C09146=1141.920,201.494,-63.208,-178.121,7.460,148.864
C09147=1141.924,201.244,-63.184,-178.124,7.457,148.864
C09148=1141.929,200.995,-63.160,-178.126,7.455,148.864
C09149=1141.933,200.747,-63.136,-178.129,7.453,148.864
C09150=1141.938,200.498,-63.112,-178.132,7.450,148.865
C09151=1141.942,200.249,-63.087,-178.135,7.448,148.865
C09152=1141.947,200.000,-63.063,-178.138,7.445,148.865
C09153=1141.951,199.752,-63.038,-178.141,7.442,148.865
C09154=1141.957,199.503,-63.015,-178.143,7.441,148.866
C09155=1141.960,199.254,-62.990,-178.146,7.438,148.866
C09156=1141.965,199.005,-62.966,-178.149,7.435,148.866
C09157=1141.969,198.757,-62.942,-178.152,7.433,148.866
C09158=1141.975,198.507,-62.918,-178.154,7.430,148.866
C09159=1141.979,198.259,-62.894,-178.158,7.428,148.867
C09160=1141.983,198.010,-62.869,-178.160,7.426,148.867
C09161=1141.987,197.761,-62.845,-178.163,7.423,148.867
C09162=1141.993,197.512,-62.821,-178.165,7.421,148.867
C09163=1141.997,197.264,-62.797,-178.169,7.418,148.868
C09164=1142.001,197.015,-62.773,-178.172,7.415,148.868
C09165=1142.006,196.766,-62.750,-178.174,7.413,148.868
C09166=1142.011,196.517,-62.725,-178.177,7.411,148.868
C09167=1142.015,196.268,-62.701,-178.180,7.408,148.868
C09168=1142.020,196.019,-62.677,-178.183,7.406,148.869
C09169=1142.024,195.771,-62.653,-178.185,7.403,148.869
C09170=1142.029,195.523,-62.629,-178.188,7.402,148.869
C09171=1142.033,195.273,-62.606,-178.191,7.399,148.869
C09172=1142.038,195.025,-62.581,-178.194,7.396,148.870
C09173=1142.042,194.775,-62.558,-178.196,7.394,148.870
C09174=1142.047,194.527,-62.533,-178.200,7.391,148.870
C09175=1142.052,194.278,-62.510,-178.202,7.389,148.870
C09176=1142.056,194.029,-62.486,-178.205,7.387,148.871
C09177=1142.061,193.780,-62.463,-178.208,7.384,148.871
C09178=1142.065,193.532,-62.439,-178.210,7.382,148.871
C09179=1142.071,193.282,-62.415,-178.213,7.379,148.871
C09180=1142.075,193.034,-62.391,-178.216,7.376,148.871
C09181=1142.080,192.785,-62.367,-178.219,7.375,148.872
C09182=1142.084,192.537,-62.343,-178.222,7.372,148.872
C09183=1142.089,192.287,-62.320,-178.224,7.370,148.872
C09184=1142.093,192.039,-62.296,-178.227,7.367,148.872
C09185=1142.097,191.789,-62.272,-178.230,7.365,148.873
C09186=1142.102,191.540,-62.249,-178.233,7.362,148.873
C09187=1142.106,191.292,-62.225,-178.236,7.360,148.873
C09188=1142.111,191.043,-62.201,-178.238,7.358,148.873
C09189=1142.115,190.794,-62.177,-178.242,7.355,148.873
C09190=1142.120,190.545,-62.154,-178.244,7.353,148.874
C09191=1142.125,190.296,-62.130,-178.247,7.351,148.874
C09192=1142.129,190.048,-62.106,-178.250,7.348,148.874
C09193=1142.134,189.799,-62.083,-178.253,7.346,148.874
C09194=1142.139,189.550,-62.060,-178.256,7.343,148.875
C09195=1142.143,189.301,-62.036,-178.258,7.341,148.875
C09196=1142.148,189.052,-62.012,-178.261,7.339,148.875
C09197=1142.152,188.803,-61.989,-178.264,7.337,148.875
C09198=1142.157,188.554,-61.965,-178.267,7.334,148.876
C09199=1142.162,188.305,-61.942,-178.269,7.332,148.876
C09200=1142.166,188.057,-61.918,-178.272,7.330,148.876
C09201=1142.171,187.808,-61.895,-178.275,7.327,148.876
C09202=1142.176,187.559,-61.871,-178.278,7.325,148.877
C09203=1142.180,187.310,-61.848,-178.281,7.322,148.877
C09204=1142.184,187.061,-61.825,-178.283,7.320,148.877
C09205=1142.189,186.813,-61.802,-178.286,7.317,148.877
C09206=1142.194,186.564,-61.778,-178.289,7.316,148.878
C09207=1142.199,186.315,-61.755,-178.292,7.313,148.878
C09208=1142.203,186.066,-61.731,-178.294,7.311,148.878
C09209=1142.208,185.817,-61.708,-178.298,7.309,148.878
C09210=1142.213,185.568,-61.685,-178.300,7.306,148.879
C09211=1142.217,185.320,-61.662,-178.303,7.304,148.879
C09212=1142.221,185.071,-61.639,-178.306,7.301,148.879
C09213=1142.226,184.821,-61.615,-178.309,7.299,148.879
C09214=1142.231,184.572,-61.592,-178.311,7.296,148.880
C09215=1142.235,184.323,-61.569,-178.314,7.295,148.880
C09216=1142.240,184.075,-61.544,-178.317,7.292,148.880
C09217=1142.244,183.806,-61.520,-178.320,7.289,148.880
C09218=1142.250,183.536,-61.495,-178.323,7.287,148.881
C09219=1142.255,183.266,-61.470,-178.326,7.285,148.881
C09220=1142.260,182.996,-61.445,-178.329,7.282,148.881
C09221=1142.264,182.748,-61.422,-178.332,7.280,148.882
C09222=1142.269,182.498,-61.399,-178.335,7.278,148.882
C09223=1142.274,182.249,-61.375,-178.337,7.276,148.882
C09224=1142.278,182.000,-61.352,-178.341,7.273,148.882
C09225=1142.283,181.752,-61.330,-178.343,7.270,148.883
C09226=1142.288,181.503,-61.306,-178.346,7.268,148.883
C09227=1142.292,181.254,-61.283,-178.349,7.266,148.883
C09228=1142.296,181.006,-61.260,-178.352,7.264,148.883
C09229=1142.301,180.757,-61.237,-178.355,7.261,148.884
C09230=1142.306,180.507,-61.214,-178.357,7.259,148.884
C09231=1142.311,180.259,-61.192,-178.360,7.257,148.884
C09232=1142.315,180.010,-61.168,-178.363,7.255,148.885
C09233=1142.320,179.761,-61.145,-178.366,7.252,148.885
C09234=1142.324,179.512,-61.122,-178.369,7.250,148.885
C09235=1142.329,179.262,-61.100,-178.371,7.248,148.885
C09236=1142.334,179.014,-61.077,-178.374,7.246,148.886
C09237=1142.338,178.765,-61.054,-178.377,7.244,148.886
C09238=1142.343,178.516,-61.031,-178.380,7.241,148.886
C09239=1142.347,178.268,-61.008,-178.382,7.239,148.886
C09240=1142.352,178.018,-60.985,-178.386,7.237,148.887
C09241=1142.357,177.770,-60.963,-178.388,7.235,148.887
C09242=1142.361,177.521,-60.939,-178.391,7.232,148.887
C09243=1142.366,177.271,-60.917,-178.393,7.230,148.887
C09244=1142.370,177.023,-60.894,-178.397,7.228,148.888
C09245=1142.376,176.774,-60.871,-178.399,7.226,148.888
C09246=1142.380,176.525,-60.849,-178.402,7.223,148.888
C09247=1142.384,176.276,-60.826,-178.405,7.221,148.889
C09248=1142.389,176.028,-60.803,-178.408,7.219,148.889
C09249=1142.394,175.778,-60.781,-178.410,7.217,148.889
C09250=1142.398,175.529,-60.758,-178.414,7.214,148.889
C09251=1142.403,175.280,-60.735,-178.416,7.212,148.890
C09252=1142.408,175.032,-60.713,-178.419,7.210,148.890
C09253=1142.412,174.783,-60.689,-178.422,7.208,148.890
C09254=1142.417,174.533,-60.667,-178.425,7.206,148.891
C09255=1142.422,174.285,-60.644,-178.427,7.203,148.891
C09256=1142.426,174.036,-60.622,-178.430,7.201,148.891
C09257=1142.431,173.787,-60.599,-178.433,7.199,148.891
C09258=1142.436,173.538,-60.577,-178.436,7.197,148.892
C09259=1142.440,173.289,-60.554,-178.439,7.194,148.892
C09260=1142.445,173.040,-60.532,-178.442,7.192,148.892
C09261=1142.449,172.792,-60.509,-178.444,7.190,148.893
C09262=1142.454,172.542,-60.487,-178.447,7.188,148.893
C09263=1142.458,172.293,-60.465,-178.450,7.186,148.893
C09264=1142.464,172.044,-60.442,-178.453,7.183,148.893
C09265=1142.468,171.795,-60.420,-178.455,7.182,148.894
C09266=1142.472,171.546,-60.397,-178.459,7.179,148.894
C09267=1142.478,171.297,-60.375,-178.461,7.177,148.894
C09268=1142.482,171.048,-60.353,-178.464,7.175,148.895
C09269=1142.486,170.800,-60.330,-178.467,7.173,148.895
C09270=1142.491,170.550,-60.308,-178.469,7.171,148.895
C09271=1142.495,170.302,-60.285,-178.472,7.168,148.895
C09272=1142.500,170.053,-60.263,-178.475,7.166,148.896
C09273=1142.505,169.803,-60.240,-178.478,7.163,148.896
C09274=1142.510,169.555,-60.219,-178.481,7.162,148.896
C09275=1142.514,169.306,-60.196,-178.483,7.160,148.897
C09276=1142.519,169.056,-60.173,-178.487,7.157,148.897
C09277=1142.524,168.808,-60.152,-178.489,7.155,148.897
C09278=1142.528,168.559,-60.129,-178.492,7.153,148.898
C09279=1142.534,168.310,-60.107,-178.495,7.151,148.898
C09280=1142.538,168.061,-60.085,-178.497,7.149,148.898
C09281=1142.543,167.812,-60.063,-178.500,7.146,148.898
C09282=1142.547,167.563,-60.041,-178.503,7.145,148.899
C09283=1142.552,167.314,-60.018,-178.506,7.142,148.899
C09284=1142.557,167.065,-59.996,-178.509,7.140,148.899
C09285=1142.561,166.816,-59.974,-178.511,7.138,148.900
C09286=1142.566,166.567,-59.952,-178.515,7.136,148.900
C09287=1142.571,166.317,-59.929,-178.517,7.134,148.900
C09288=1142.576,166.069,-59.908,-178.519,7.132,148.901
C09289=1142.580,165.820,-59.885,-178.523,7.130,148.901
C09290=1142.584,165.571,-59.863,-178.525,7.128,148.901
C09291=1142.589,165.322,-59.841,-178.528,7.125,148.901
C09292=1142.594,165.073,-59.820,-178.531,7.123,148.902
C09293=1142.599,164.824,-59.797,-178.534,7.122,148.902
C09294=1142.603,164.575,-59.775,-178.537,7.119,148.903
C09295=1142.608,164.326,-59.753,-178.539,7.117,148.903
C09296=1142.613,164.077,-59.732,-178.542,7.115,148.903
C09297=1142.617,163.829,-59.710,-178.545,7.113,148.903
C09298=1142.622,163.579,-59.688,-178.548,7.111,148.904
C09299=1142.627,163.331,-59.666,-178.551,7.108,148.904
C09300=1142.631,163.081,-59.644,-178.553,7.106,148.904
C09301=1142.636,162.832,-59.622,-178.556,7.105,148.905
C09302=1142.641,162.583,-59.600,-178.559,7.102,148.905
C09303=1142.646,162.334,-59.578,-178.562,7.100,148.905
C09304=1142.650,162.085,-59.556,-178.564,7.098,148.906
C09305=1142.655,161.836,-59.534,-178.568,7.096,148.906
C09306=1142.659,161.587,-59.512,-178.570,7.094,148.906
C09307=1142.664,161.338,-59.491,-178.573,7.092,148.906
C09308=1142.669,161.090,-59.469,-178.576,7.089,148.907
C09309=1142.673,160.840,-59.447,-178.579,7.088,148.907
C09310=1142.678,160.591,-59.426,-178.581,7.086,148.908
C09311=1142.682,160.342,-59.404,-178.584,7.083,148.908
C09312=1142.687,160.093,-59.382,-178.587,7.081,148.908
C09313=1142.692,159.844,-59.360,-178.590,7.080,148.908
C09314=1142.696,159.595,-59.338,-178.593,7.077,148.909
C09315=1142.701,159.346,-59.317,-178.596,7.075,148.909
C09316=1142.706,159.096,-59.295,-178.598,7.073,148.909
C09317=1142.711,158.848,-59.274,-178.601,7.071,148.910
C09318=1142.716,158.599,-59.252,-178.604,7.069,148.910
C09319=1142.720,158.350,-59.230,-178.607,7.067,148.910
C09320=1142.725,158.101,-59.208,-178.610,7.065,148.911
C09321=1142.729,157.832,-59.186,-178.613,7.063,148.911
C09322=1142.735,157.563,-59.162,-178.615,7.060,148.911
C09323=1142.740,157.294,-59.139,-178.618,7.059,148.912
C09324=1142.745,157.025,-59.115,-178.621,7.056,148.912
C09325=1142.750,156.776,-59.094,-178.624,7.054,148.912
C09326=1142.755,156.527,-59.073,-178.627,7.052,148.913
C09327=1142.758,156.278,-59.051,-178.630,7.050,148.913
C09328=1142.764,156.029,-59.030,-178.633,7.048,148.914
C09329=1142.769,155.780,-59.009,-178.636,7.045,148.914
C09330=1142.773,155.531,-58.987,-178.638,7.044,148.914
C09331=1142.778,155.282,-58.966,-178.641,7.042,148.915
C09332=1142.783,155.033,-58.944,-178.644,7.040,148.915
C09333=1142.788,154.784,-58.922,-178.647,7.038,148.915
C09334=1142.792,154.535,-58.902,-178.649,7.036,148.915
C09335=1142.796,154.286,-58.880,-178.652,7.034,148.916
C09336=1142.802,154.037,-58.859,-178.655,7.031,148.916
C09337=1142.806,153.787,-58.837,-178.658,7.030,148.917
C09338=1142.811,153.538,-58.816,-178.661,7.028,148.917
C09339=1142.816,153.290,-58.794,-178.663,7.026,148.917
C09340=1142.820,153.041,-58.774,-178.666,7.023,148.917
C09341=1142.825,152.792,-58.752,-178.669,7.022,148.918
C09342=1142.830,152.542,-58.731,-178.672,7.020,148.918
C09343=1142.835,152.293,-58.709,-178.675,7.017,148.919
C09344=1142.839,152.044,-58.689,-178.678,7.016,148.919
C09345=1142.844,151.796,-58.667,-178.680,7.014,148.919
C09346=1142.849,151.546,-58.646,-178.683,7.012,148.920
C09347=1142.853,151.297,-58.624,-178.686,7.009,148.920
C09348=1142.858,151.048,-58.604,-178.689,7.008,148.920
C09349=1142.863,150.799,-58.583,-178.691,7.006,148.921
C09350=1142.868,150.550,-58.561,-178.694,7.004,148.921
C09351=1142.872,150.301,-58.540,-178.697,7.002,148.921
C09352=1142.877,150.052,-58.519,-178.700,7.000,148.922
C09353=1142.882,149.803,-58.498,-178.702,6.998,148.922
C09354=1142.886,149.554,-58.477,-178.705,6.996,148.922
C09355=1142.891,149.305,-58.456,-178.708,6.994,148.923
C09356=1142.896,149.056,-58.435,-178.711,6.992,148.923
C09357=1142.900,148.806,-58.414,-178.714,6.990,148.923
C09358=1142.905,148.558,-58.392,-178.716,6.989,148.924
C09359=1142.910,148.308,-58.371,-178.720,6.986,148.924
C09360=1142.915,148.059,-58.351,-178.722,6.984,148.924
C09361=1142.920,147.810,-58.330,-178.725,6.982,148.925
C09362=1142.925,147.561,-58.308,-178.727,6.981,148.925
C09363=1142.929,147.313,-58.288,-178.731,6.978,148.926
C09364=1142.934,147.063,-58.266,-178.733,6.976,148.926
C09365=1142.938,146.814,-58.246,-178.736,6.975,148.926
C09366=1142.943,146.565,-58.224,-178.739,6.973,148.927
C09367=1142.947,146.316,-58.204,-178.742,6.970,148.927
C09368=1142.953,146.067,-58.183,-178.745,6.969,148.927
C09369=1142.958,145.818,-58.162,-178.747,6.967,148.928
C09370=1142.962,145.569,-58.142,-178.750,6.965,148.928
C09371=1142.967,145.319,-58.121,-178.752,6.963,148.928
C09372=1142.971,145.071,-58.100,-178.756,6.961,148.929
C09373=1142.977,144.822,-58.079,-178.758,6.959,148.929
C09374=1142.980,144.572,-58.058,-178.761,6.957,148.930
C09375=1142.986,144.323,-58.037,-178.764,6.956,148.930
C09376=1142.990,144.074,-58.017,-178.767,6.953,148.930
C09377=1142.995,143.825,-57.996,-178.770,6.951,148.931
C09378=1143.000,143.576,-57.975,-178.772,6.949,148.931
C09379=1143.005,143.326,-57.954,-178.775,6.948,148.931
C09380=1143.009,143.077,-57.934,-178.778,6.946,148.932
C09381=1143.014,142.828,-57.913,-178.781,6.943,148.932
C09382=1143.019,142.579,-57.893,-178.784,6.942,148.932
C09383=1143.023,142.330,-57.872,-178.786,6.940,148.933
C09384=1143.028,142.081,-57.851,-178.789,6.938,148.933
C09385=1143.033,141.832,-57.831,-178.792,6.937,148.934
C09386=1143.038,141.583,-57.810,-178.795,6.934,148.934
C09387=1143.043,141.334,-57.790,-178.798,6.932,148.934
C09388=1143.047,141.085,-57.769,-178.800,6.931,148.935
C09389=1143.052,140.836,-57.748,-178.803,6.929,148.935
C09390=1143.057,140.587,-57.728,-178.805,6.927,148.935
C09391=1143.062,140.337,-57.707,-178.808,6.925,148.936
C09392=1143.066,140.089,-57.687,-178.811,6.923,148.936
C09393=1143.071,139.840,-57.666,-178.814,6.921,148.936
C09394=1143.076,139.590,-57.645,-178.817,6.919,148.937
C09395=1143.081,139.341,-57.626,-178.820,6.917,148.937
C09396=1143.085,139.092,-57.605,-178.822,6.916,148.938
C09397=1143.090,138.843,-57.584,-178.825,6.914,148.938
C09398=1143.095,138.594,-57.564,-178.828,6.912,148.938
C09399=1143.099,138.345,-57.543,-178.831,6.910,148.939
C09400=1143.104,138.095,-57.522,-178.834,6.908,148.939
C09401=1143.109,137.846,-57.503,-178.837,6.906,148.940
C09402=1143.113,137.597,-57.482,-178.839,6.905,148.940
C09403=1143.118,137.348,-57.462,-178.842,6.903,148.940
C09404=1143.123,137.099,-57.441,-178.845,6.901,148.941
C09405=1143.128,136.850,-57.421,-178.848,6.899,148.941
C09406=1143.133,136.601,-57.401,-178.851,6.897,148.941
C09407=1143.138,136.352,-57.380,-178.853,6.895,148.942
C09408=1143.142,136.103,-57.360,-178.856,6.893,148.942
C09409=1143.147,135.853,-57.340,-178.858,6.892,148.942
C09410=1143.152,135.604,-57.320,-178.861,6.890,148.943
C09411=1143.156,135.355,-57.300,-178.864,6.887,148.943
C09412=1143.161,135.106,-57.279,-178.867,6.886,148.944
C09413=1143.166,134.856,-57.259,-178.870,6.884,148.944
C09414=1143.170,134.607,-57.239,-178.873,6.882,148.944
C09415=1143.176,134.359,-57.219,-178.875,6.881,148.945
C09416=1143.180,134.110,-57.199,-178.878,6.879,148.945
C09417=1143.185,133.860,-57.178,-178.881,6.877,148.946
C09418=1143.190,133.611,-57.158,-178.884,6.875,148.946
C09419=1143.195,133.362,-57.138,-178.887,6.873,148.946
C09420=1143.199,133.112,-57.118,-178.889,6.871,148.947
C09421=1143.204,132.864,-57.098,-178.892,6.870,148.947
C09422=1143.209,132.615,-57.078,-178.895,6.868,148.948
C09423=1143.214,132.365,-57.058,-178.898,6.866,148.948
C09424=1143.219,132.116,-57.037,-178.900,6.864,148.948
C09425=1143.224,131.848,-57.016,-178.904,6.862,148.949
C09426=1143.229,131.579,-56.995,-178.906,6.860,148.949
C09427=1143.234,131.311,-56.973,-178.909,6.859,148.949
C09428=1143.239,131.042,-56.952,-178.912,6.856,148.950
C09429=1143.243,130.792,-56.932,-178.915,6.854,148.950
C09430=1143.249,130.544,-56.912,-178.918,6.853,148.951
C09431=1143.254,130.294,-56.892,-178.921,6.851,148.951
C09432=1143.258,130.045,-56.871,-178.923,6.849,148.951
C09433=1143.263,129.796,-56.852,-178.926,6.848,148.952
C09434=1143.268,129.547,-56.831,-178.929,6.846,148.952
C09435=1143.273,129.298,-56.812,-178.931,6.844,148.953
C09436=1143.278,129.048,-56.793,-178.935,6.842,148.953
C09437=1143.282,128.799,-56.772,-178.937,6.840,148.953
C09438=1143.287,128.550,-56.752,-178.940,6.838,148.954
C09439=1143.292,128.302,-56.732,-178.943,6.837,148.954
C09440=1143.297,128.052,-56.713,-178.946,6.835,148.955
C09441=1143.301,127.802,-56.693,-178.949,6.834,148.955
C09442=1143.306,127.553,-56.673,-178.952,6.832,148.956
C09443=1143.311,127.305,-56.653,-178.954,6.830,148.956
C09444=1143.316,127.055,-56.634,-178.957,6.828,148.956
C09445=1143.320,126.806,-56.613,-178.960,6.827,148.957
C09446=1143.326,126.557,-56.594,-178.962,6.825,148.957
C09447=1143.330,126.308,-56.575,-178.965,6.823,148.958
C09448=1143.335,126.058,-56.555,-178.968,6.822,148.958
C09449=1143.339,125.809,-56.535,-178.971,6.819,148.958
C09450=1143.344,125.561,-56.516,-178.974,6.817,148.959
C09451=1143.349,125.311,-56.496,-178.977,6.816,148.959
C09452=1143.354,125.061,-56.476,-178.979,6.814,148.960
C09453=1143.359,124.813,-56.456,-178.982,6.812,148.960
C09454=1143.364,124.564,-56.437,-178.985,6.811,148.960
C09455=1143.368,124.314,-56.417,-178.987,6.809,148.961
C09456=1143.374,124.065,-56.398,-178.990,6.807,148.961
C09457=1143.378,123.816,-56.378,-178.993,6.806,148.962
C09458=1143.382,123.566,-56.359,-178.996,6.804,148.962
C09459=1143.387,123.318,-56.339,-178.998,6.802,148.962
C09460=1143.392,123.069,-56.319,-179.001,6.800,148.963
C09461=1143.397,122.819,-56.300,-179.004,6.799,148.963
C09462=1143.402,122.570,-56.281,-179.007,6.797,148.964
C09463=1143.407,122.321,-56.261,-179.009,6.795,148.964
C09464=1143.412,122.072,-56.242,-179.012,6.794,148.964
C09465=1143.416,121.822,-56.223,-179.015,6.792,148.965
C09466=1143.421,121.573,-56.203,-179.017,6.790,148.965
C09467=1143.426,121.324,-56.184,-179.020,6.789,148.966
C09468=1143.431,121.074,-56.164,-179.023,6.787,148.966
C09469=1143.435,120.825,-56.145,-179.026,6.785,148.966
C09470=1143.440,120.576,-56.126,-179.029,6.783,148.967
C09471=1143.445,120.327,-56.106,-179.032,6.781,148.967
C09472=1143.451,120.078,-56.087,-179.035,6.780,148.968
C09473=1143.455,119.829,-56.068,-179.038,6.778,148.968
C09474=1143.460,119.580,-56.048,-179.040,6.776,148.969
C09475=1143.465,119.330,-56.029,-179.043,6.775,148.969
C09476=1143.469,119.081,-56.009,-179.046,6.773,148.969
C09477=1143.474,118.832,-55.990,-179.048,6.771,148.970
C09478=1143.479,118.582,-55.971,-179.051,6.770,148.970
C09479=1143.484,118.334,-55.951,-179.054,6.768,148.971
C09480=1143.488,118.084,-55.932,-179.057,6.766,148.971
C09481=1143.493,117.835,-55.913,-179.059,6.764,148.971
C09482=1143.498,117.586,-55.893,-179.062,6.763,148.972
C09483=1143.503,117.337,-55.875,-179.065,6.761,148.972
C09484=1143.508,117.087,-55.856,-179.068,6.759,148.973
C09485=1143.513,116.838,-55.836,-179.071,6.758,148.973
C09486=1143.517,116.589,-55.817,-179.073,6.756,148.974
C09487=1143.523,116.340,-55.798,-179.076,6.755,148.974
C09488=1143.527,116.091,-55.778,-179.079,6.753,148.974
C09489=1143.532,115.842,-55.760,-179.082,6.751,148.975
C09490=1143.537,115.592,-55.741,-179.084,6.750,148.975
C09491=1143.542,115.343,-55.721,-179.087,6.748,148.976
C09492=1143.546,115.094,-55.702,-179.090,6.746,148.976
C09493=1143.552,114.845,-55.683,-179.093,6.745,148.977
C09494=1143.556,114.595,-55.665,-179.095,6.743,148.977
C09495=1143.561,114.346,-55.645,-179.098,6.741,148.977
C09496=1143.565,114.097,-55.626,-179.101,6.739,148.978
C09497=1143.571,113.848,-55.607,-179.104,6.738,148.978
C09498=1143.576,113.598,-55.588,-179.107,6.736,148.979
C09499=1143.580,113.349,-55.569,-179.109,6.736,148.979
C09500=1143.585,113.100,-55.550,-179.112,6.734,148.980
C09501=1143.590,112.850,-55.532,-179.114,6.732,148.980
C09502=1143.595,112.601,-55.512,-179.117,6.730,148.980
C09503=1143.599,112.352,-55.493,-179.120,6.729,148.981
C09504=1143.605,112.103,-55.475,-179.122,6.727,148.981
C09505=1143.609,111.854,-55.456,-179.125,6.725,148.982
C09506=1143.614,111.605,-55.437,-179.128,6.724,148.982
C09507=1143.619,111.355,-55.418,-179.131,6.722,148.983
C09508=1143.624,111.106,-55.399,-179.134,6.721,148.983
C09509=1143.629,110.857,-55.381,-179.137,6.719,148.983
C09510=1143.634,110.607,-55.361,-179.139,6.717,148.984
C09511=1143.639,110.358,-55.343,-179.142,6.716,148.984
C09512=1143.643,110.109,-55.324,-179.145,6.714,148.985
C09513=1143.648,109.860,-55.305,-179.147,6.712,148.985
C09514=1143.654,109.610,-55.286,-179.150,6.711,148.986
C09515=1143.658,109.361,-55.267,-179.153,6.709,148.986
C09516=1143.662,109.112,-55.249,-179.156,6.708,148.987
C09517=1143.668,108.863,-55.230,-179.159,6.706,148.987
C09518=1143.672,108.613,-55.212,-179.162,6.704,148.987
C09519=1143.677,108.364,-55.192,-179.164,6.703,148.988
C09520=1143.682,108.115,-55.174,-179.166,6.702,148.988
C09521=1143.686,107.866,-55.155,-179.169,6.700,148.989
C09522=1143.692,107.617,-55.137,-179.172,6.698,148.989
C09523=1143.696,107.367,-55.118,-179.175,6.697,148.990
C09524=1143.701,107.118,-55.100,-179.178,6.695,148.990
C09525=1143.707,106.869,-55.081,-179.181,6.694,148.990
C09526=1143.711,106.619,-55.062,-179.183,6.692,148.991
C09527=1143.716,106.370,-55.044,-179.186,6.690,148.991
C09528=1143.721,106.121,-55.026,-179.189,6.689,148.992
C09529=1143.726,105.853,-55.005,-179.192,6.687,148.992
C09530=1143.731,105.584,-54.985,-179.195,6.686,148.993
C09531=1143.736,105.316,-54.966,-179.197,6.684,148.993
C09532=1143.742,105.047,-54.946,-179.200,6.682,148.994
C09533=1143.747,104.798,-54.927,-179.203,6.681,148.994
C09534=1143.751,104.549,-54.909,-179.206,6.679,148.995
C09535=1143.757,104.299,-54.890,-179.209,6.677,148.995
C09536=1143.761,104.050,-54.871,-179.212,6.676,148.995
C09537=1143.766,103.801,-54.853,-179.214,6.674,148.996
C09538=1143.770,103.551,-54.835,-179.217,6.672,148.996
C09539=1143.776,103.303,-54.816,-179.220,6.671,148.997
C09540=1143.781,103.053,-54.798,-179.223,6.669,148.997
C09541=1143.786,102.804,-54.780,-179.225,6.669,148.998
C09542=1143.790,102.554,-54.761,-179.228,6.667,148.998
C09543=1143.796,102.305,-54.743,-179.231,6.665,148.999
C09544=1143.800,102.056,-54.724,-179.233,6.663,148.999
C09545=1143.805,101.807,-54.706,-179.236,6.662,148.999
C09546=1143.809,101.557,-54.688,-179.239,6.660,149.000
C09547=1143.814,101.308,-54.670,-179.242,6.659,149.000
C09548=1143.820,101.059,-54.651,-179.245,6.657,149.001
C09549=1143.825,100.809,-54.633,-179.247,6.655,149.001
C09550=1143.829,100.561,-54.615,-179.250,6.655,149.002
C09551=1143.834,100.311,-54.596,-179.252,6.653,149.002
C09552=1143.839,100.062,-54.578,-179.256,6.652,149.003
C09553=1143.844,99.813,-54.560,-179.258,6.650,149.003
C09554=1143.849,99.563,-54.542,-179.261,6.648,149.004
C09555=1143.854,99.314,-54.524,-179.264,6.647,149.004
C09556=1143.858,99.064,-54.505,-179.267,6.645,149.004
C09557=1143.863,98.815,-54.487,-179.269,6.644,149.005
C09558=1143.868,98.566,-54.469,-179.272,6.643,149.005
C09559=1143.873,98.317,-54.451,-179.275,6.641,149.006
C09560=1143.878,98.067,-54.433,-179.277,6.639,149.006
C09561=1143.883,97.818,-54.416,-179.280,6.638,149.007
C09562=1143.887,97.568,-54.397,-179.283,6.636,149.007
C09563=1143.892,97.319,-54.379,-179.286,6.635,149.008
C09564=1143.897,97.070,-54.361,-179.288,6.634,149.008
C09565=1143.903,96.820,-54.343,-179.291,6.632,149.009
C09566=1143.908,96.571,-54.325,-179.294,6.630,149.009
C09567=1143.913,96.322,-54.307,-179.296,6.629,149.009
C09568=1143.918,96.073,-54.289,-179.300,6.627,149.010
C09569=1143.922,95.824,-54.271,-179.302,6.626,149.011
C09570=1143.927,95.574,-54.252,-179.305,6.624,149.011
C09571=1143.932,95.325,-54.234,-179.307,6.623,149.011
C09572=1143.937,95.076,-54.216,-179.310,6.622,149.012
C09573=1143.942,94.826,-54.198,-179.313,6.620,149.012
C09574=1143.946,94.577,-54.180,-179.316,6.619,149.013
C09575=1143.951,94.328,-54.162,-179.319,6.617,149.013
C09576=1143.956,94.079,-54.144,-179.321,6.616,149.014
C09577=1143.961,93.829,-54.127,-179.323,6.614,149.014
C09578=1143.966,93.580,-54.109,-179.326,6.613,149.015
C09579=1143.971,93.331,-54.091,-179.329,6.611,149.015
C09580=1143.976,93.082,-54.073,-179.332,6.610,149.016
C09581=1143.980,92.833,-54.056,-179.335,6.608,149.016
C09582=1143.986,92.583,-54.039,-179.337,6.607,149.016
C09583=1143.990,92.333,-54.020,-179.340,6.606,149.017
C09584=1143.995,92.084,-54.002,-179.343,6.604,149.017
C09585=1144.000,91.835,-53.984,-179.346,6.602,149.018
C09586=1144.005,91.585,-53.966,-179.348,6.601,149.018
C09587=1144.010,91.336,-53.949,-179.351,6.600,149.019
C09588=1144.015,91.086,-53.931,-179.354,6.599,149.019
C09589=1144.020,90.837,-53.913,-179.357,6.597,149.020
C09590=1144.025,90.588,-53.895,-179.359,6.595,149.020
C09591=1144.029,90.339,-53.878,-179.362,6.594,149.021
C09592=1144.034,90.089,-53.860,-179.364,6.593,149.021
C09593=1144.039,89.840,-53.843,-179.367,6.591,149.022
C09594=1144.044,89.591,-53.825,-179.370,6.590,149.022
C09595=1144.049,89.341,-53.807,-179.373,6.588,149.023
C09596=1144.054,89.092,-53.789,-179.376,6.586,149.023
C09597=1144.059,88.842,-53.772,-179.378,6.586,149.024
C09598=1144.063,88.594,-53.755,-179.381,6.584,149.024
C09599=1144.068,88.344,-53.737,-179.384,6.583,149.024
C09600=1144.073,88.095,-53.719,-179.386,6.581,149.025
C09601=1144.078,87.845,-53.701,-179.389,6.579,149.025
C09602=1144.084,87.596,-53.684,-179.392,6.579,149.026
C09603=1144.088,87.347,-53.667,-179.395,6.577,149.026
C09604=1144.094,87.098,-53.650,-179.397,6.575,149.027
C09605=1144.099,86.848,-53.632,-179.400,6.574,149.027
C09606=1144.103,86.599,-53.614,-179.403,6.573,149.028
C09607=1144.108,86.350,-53.597,-179.405,6.572,149.028
C09608=1144.113,86.101,-53.579,-179.408,6.570,149.029
C09609=1144.118,85.851,-53.562,-179.411,6.568,149.029
C09610=1144.123,85.602,-53.544,-179.413,6.568,149.030
C09611=1144.127,85.352,-53.527,-179.416,6.566,149.030
C09612=1144.132,85.103,-53.509,-179.419,6.564,149.031
C09613=1144.138,84.853,-53.492,-179.422,6.563,149.031
C09614=1144.142,84.604,-53.475,-179.425,6.561,149.032
C09615=1144.147,84.355,-53.457,-179.427,6.561,149.032
C09616=1144.152,84.105,-53.440,-179.430,6.559,149.033
C09617=1144.158,83.856,-53.423,-179.433,6.557,149.033
C09618=1144.162,83.607,-53.406,-179.435,6.555,149.033
C09619=1144.167,83.358,-53.388,-179.438,6.555,149.034
C09620=1144.172,83.108,-53.371,-179.441,6.553,149.035
C09621=1144.176,82.859,-53.353,-179.443,6.552,149.035
C09622=1144.182,82.609,-53.336,-179.446,6.551,149.035
C09623=1144.186,82.360,-53.319,-179.449,6.549,149.036
C09624=1144.191,82.110,-53.301,-179.452,6.548,149.036
C09625=1144.197,81.861,-53.284,-179.454,6.546,149.037
C09626=1144.201,81.612,-53.268,-179.457,6.546,149.038
C09627=1144.206,81.363,-53.250,-179.460,6.544,149.038
C09628=1144.211,81.113,-53.233,-179.462,6.542,149.038
C09629=1144.216,80.863,-53.216,-179.465,6.541,149.039
C09630=1144.221,80.614,-53.198,-179.468,6.540,149.039
C09631=1144.226,80.365,-53.182,-179.470,6.539,149.040
C09632=1144.231,80.116,-53.164,-179.473,6.537,149.040
C09633=1144.237,79.847,-53.146,-179.476,6.535,149.041
C09634=1144.242,79.579,-53.128,-179.479,6.534,149.041
C09635=1144.247,79.311,-53.108,-179.482,6.532,149.042
C09636=1144.252,79.042,-53.090,-179.485,6.531,149.042
C09637=1144.257,78.793,-53.073,-179.487,6.530,149.043
C09638=1144.263,78.543,-53.056,-179.490,6.528,149.043
C09639=1144.267,78.294,-53.040,-179.493,6.527,149.044
C09640=1144.272,78.045,-53.022,-179.495,6.526,149.044
C09641=1144.276,77.795,-53.005,-179.498,6.525,149.045
C09642=1144.282,77.546,-52.988,-179.501,6.523,149.045
C09643=1144.287,77.297,-52.971,-179.504,6.522,149.046
C09644=1144.292,77.047,-52.954,-179.506,6.521,149.046
C09645=1144.296,76.797,-52.937,-179.509,6.519,149.047
C09646=1144.302,76.548,-52.921,-179.512,6.518,149.047
C09647=1144.306,76.299,-52.903,-179.514,6.517,149.048
C09648=1144.311,76.050,-52.886,-179.517,6.515,149.048
C09649=1144.316,75.800,-52.869,-179.520,6.514,149.049
C09650=1144.321,75.551,-52.853,-179.523,6.513,149.049
C09651=1144.326,75.301,-52.836,-179.525,6.511,149.050
C09652=1144.331,75.052,-52.819,-179.528,6.510,149.050
C09653=1144.336,74.802,-52.802,-179.530,6.509,149.051
C09654=1144.341,74.553,-52.785,-179.533,6.508,149.051
C09655=1144.346,74.304,-52.769,-179.536,6.506,149.052
C09656=1144.351,74.054,-52.751,-179.538,6.505,149.052
C09657=1144.356,73.805,-52.735,-179.541,6.504,149.053
C09658=1144.361,73.556,-52.718,-179.544,6.502,149.053
C09659=1144.366,73.306,-52.701,-179.546,6.501,149.054
C09660=1144.371,73.057,-52.685,-179.549,6.500,149.054
C09661=1144.376,72.807,-52.668,-179.552,6.498,149.055
C09662=1144.380,72.558,-52.651,-179.555,6.497,149.055
C09663=1144.386,72.309,-52.634,-179.557,6.496,149.056
C09664=1144.391,72.059,-52.617,-179.560,6.495,149.056
C09665=1144.395,71.810,-52.601,-179.563,6.494,149.057
C09666=1144.401,71.561,-52.584,-179.565,6.492,149.057
C09667=1144.406,71.311,-52.567,-179.569,6.491,149.058
C09668=1144.410,71.062,-52.551,-179.571,6.490,149.058
C09669=1144.416,70.813,-52.534,-179.573,6.488,149.059
C09670=1144.420,70.563,-52.517,-179.576,6.487,149.059
C09671=1144.425,70.314,-52.500,-179.579,6.486,149.060
C09672=1144.430,70.064,-52.485,-179.582,6.484,149.060
C09673=1144.435,69.815,-52.467,-179.584,6.483,149.061
C09674=1144.440,69.565,-52.451,-179.587,6.482,149.061
C09675=1144.445,69.316,-52.434,-179.590,6.481,149.062
C09676=1144.450,69.067,-52.417,-179.592,6.479,149.062
C09677=1144.455,68.818,-52.401,-179.595,6.478,149.063
C09678=1144.460,68.568,-52.385,-179.598,6.477,149.063
C09679=1144.465,68.318,-52.368,-179.601,6.475,149.064
C09680=1144.470,68.069,-52.351,-179.603,6.474,149.064
C09681=1144.475,67.820,-52.335,-179.606,6.473,149.065
C09682=1144.480,67.571,-52.318,-179.608,6.472,149.065
C09683=1144.485,67.321,-52.302,-179.611,6.470,149.066
C09684=1144.489,67.071,-52.286,-179.614,6.469,149.066
C09685=1144.495,66.822,-52.269,-179.616,6.468,149.067
C09686=1144.499,66.573,-52.252,-179.619,6.467,149.067
C09687=1144.505,66.323,-52.237,-179.622,6.465,149.068
C09688=1144.509,66.074,-52.220,-179.624,6.465,149.068
C09689=1144.514,65.825,-52.204,-179.627,6.463,149.069
C09690=1144.519,65.575,-52.188,-179.630,6.462,149.069
C09691=1144.524,65.325,-52.170,-179.633,6.461,149.070
C09692=1144.530,65.076,-52.154,-179.635,6.459,149.070
C09693=1144.534,64.826,-52.138,-179.638,6.459,149.071
C09694=1144.539,64.577,-52.122,-179.641,6.457,149.071
C09695=1144.544,64.328,-52.105,-179.643,6.456,149.072
C09696=1144.549,64.078,-52.090,-179.646,6.454,149.072
C09697=1144.554,63.829,-52.073,-179.649,6.453,149.073
C09698=1144.560,63.580,-52.056,-179.651,6.452,149.073
C09699=1144.564,63.330,-52.040,-179.654,6.451,149.074
C09700=1144.569,63.081,-52.024,-179.656,6.450,149.074
C09701=1144.574,62.831,-52.008,-179.659,6.449,149.075
C09702=1144.579,62.582,-51.992,-179.662,6.447,149.075
C09703=1144.584,62.332,-51.976,-179.664,6.446,149.076
C09704=1144.589,62.083,-51.959,-179.667,6.445,149.076
C09705=1144.594,61.834,-51.943,-179.669,6.444,149.077
C09706=1144.599,61.584,-51.927,-179.673,6.443,149.078
C09707=1144.604,61.335,-51.910,-179.675,6.441,149.078
C09708=1144.609,61.085,-51.895,-179.678,6.440,149.078
C09709=1144.613,60.836,-51.878,-179.681,6.439,149.079
C09710=1144.619,60.587,-51.862,-179.683,6.438,149.079
C09711=1144.623,60.337,-51.846,-179.686,6.436,149.080
C09712=1144.629,60.088,-51.830,-179.689,6.435,149.081
C09713=1144.634,59.839,-51.814,-179.691,6.434,149.081
C09714=1144.638,59.589,-51.798,-179.694,6.433,149.081
C09715=1144.644,59.339,-51.782,-179.696,6.432,149.082
C09716=1144.648,59.090,-51.766,-179.699,6.430,149.083
C09717=1144.654,58.841,-51.750,-179.701,6.430,149.083
C09718=1144.658,58.591,-51.733,-179.705,6.428,149.084
C09719=1144.664,58.342,-51.718,-179.707,6.427,149.084
C09720=1144.669,58.093,-51.702,-179.709,6.426,149.085
C09721=1144.673,57.843,-51.686,-179.713,6.425,149.085
C09722=1144.679,57.593,-51.670,-179.715,6.424,149.086
C09723=1144.683,57.344,-51.653,-179.718,6.422,149.086
C09724=1144.689,57.094,-51.638,-179.720,6.422,149.087
C09725=1144.694,56.845,-51.622,-179.723,6.420,149.087
C09726=1144.699,56.596,-51.606,-179.725,6.419,149.088
C09727=1144.704,56.346,-51.590,-179.728,6.418,149.088
C09728=1144.709,56.096,-51.574,-179.731,6.416,149.089
C09729=1144.714,55.847,-51.558,-179.733,6.415,149.089
C09730=1144.719,55.598,-51.542,-179.737,6.414,149.090
C09731=1144.723,55.348,-51.527,-179.739,6.413,149.090
C09732=1144.729,55.099,-51.511,-179.742,6.412,149.091
C09733=1144.734,54.850,-51.495,-179.744,6.411,149.091
C09734=1144.739,54.600,-51.479,-179.747,6.409,149.092
C09735=1144.744,54.350,-51.463,-179.749,6.409,149.092
C09736=1144.749,54.101,-51.448,-179.752,6.407,149.093
C09737=1144.754,53.832,-51.430,-179.755,6.406,149.093
C09738=1144.760,53.563,-51.413,-179.758,6.405,149.094
C09739=1144.765,53.295,-51.396,-179.761,6.404,149.095
C09740=1144.770,53.027,-51.380,-179.764,6.402,149.095
C09741=1144.776,52.777,-51.364,-179.766,6.401,149.096
C09742=1144.780,52.528,-51.348,-179.769,6.400,149.096
C09743=1144.785,52.278,-51.332,-179.771,6.399,149.097
C09744=1144.791,52.029,-51.316,-179.774,6.398,149.097
C09745=1144.795,51.779,-51.301,-179.777,6.397,149.098
C09746=1144.800,51.530,-51.285,-179.779,6.395,149.098
C09747=1144.806,51.280,-51.270,-179.782,6.395,149.099
C09748=1144.810,51.030,-51.254,-179.785,6.393,149.099
C09749=1144.816,50.782,-51.238,-179.787,6.393,149.100
C09750=1144.820,50.532,-51.223,-179.790,6.391,149.100
C09751=1144.826,50.283,-51.207,-179.792,6.390,149.101
C09752=1144.830,50.033,-51.191,-179.795,6.389,149.101
C09753=1144.836,49.784,-51.176,-179.798,6.388,149.102
C09754=1144.840,49.534,-51.161,-179.800,6.387,149.102
C09755=1144.846,49.285,-51.145,-179.803,6.386,149.103
C09756=1144.851,49.035,-51.129,-179.806,6.385,149.104
C09757=1144.855,48.786,-51.114,-179.808,6.384,149.104
C09758=1144.861,48.536,-51.098,-179.811,6.382,149.105
C09759=1144.865,48.286,-51.082,-179.813,6.382,149.105
C09760=1144.870,48.037,-51.067,-179.816,6.380,149.106
C09761=1144.875,47.788,-51.052,-179.819,6.379,149.106
C09762=1144.881,47.538,-51.036,-179.821,6.378,149.107
C09763=1144.885,47.289,-51.021,-179.824,6.377,149.107
C09764=1144.890,47.039,-51.005,-179.827,6.376,149.108
C09765=1144.896,46.790,-50.990,-179.829,6.375,149.108
C09766=1144.900,46.541,-50.975,-179.832,6.374,149.109
C09767=1144.906,46.291,-50.959,-179.834,6.373,149.109
C09768=1144.911,46.042,-50.944,-179.837,6.371,149.110
C09769=1144.915,45.792,-50.928,-179.840,6.371,149.111
C09770=1144.920,45.543,-50.913,-179.843,6.369,149.111
C09771=1144.926,45.293,-50.897,-179.845,6.368,149.111
C09772=1144.931,45.044,-50.883,-179.848,6.367,149.112
C09773=1144.936,44.794,-50.867,-179.850,6.366,149.113
C09774=1144.940,44.544,-50.852,-179.853,6.364,149.113
C09775=1144.946,44.295,-50.836,-179.856,6.364,149.114
C09776=1144.951,44.046,-50.821,-179.858,6.362,149.114
C09777=1144.956,43.797,-50.806,-179.861,6.362,149.115
C09778=1144.961,43.547,-50.790,-179.864,6.360,149.115
C09779=1144.966,43.297,-50.776,-179.866,6.359,149.116
C09780=1144.971,43.047,-50.760,-179.868,6.359,149.116
C09781=1144.975,42.798,-50.745,-179.871,6.357,149.117
C09782=1144.981,42.549,-50.729,-179.874,6.357,149.117
C09783=1144.986,42.300,-50.714,-179.877,6.355,149.118
C09784=1144.991,42.050,-50.699,-179.879,6.354,149.118
C09785=1144.997,41.800,-50.684,-179.882,6.353,149.119
C09786=1145.001,41.551,-50.669,-179.884,6.352,149.119
C09787=1145.007,41.302,-50.653,-179.887,6.351,149.120
C09788=1145.011,41.051,-50.639,-179.890,6.350,149.121
C09789=1145.016,40.802,-50.623,-179.892,6.349,149.121
C09790=1145.021,40.553,-50.608,-179.895,6.348,149.122
C09791=1145.026,40.304,-50.592,-179.897,6.347,149.122
C09792=1145.031,40.054,-50.578,-179.900,6.346,149.123
C09793=1145.037,39.804,-50.563,-179.903,6.345,149.123
C09794=1145.041,39.555,-50.548,-179.905,6.343,149.124
C09795=1145.046,39.306,-50.533,-179.908,6.343,149.124
C09796=1145.052,39.056,-50.518,-179.911,6.341,149.125
C09797=1145.056,38.807,-50.503,-179.913,6.341,149.125
C09798=1145.062,38.557,-50.488,-179.916,6.340,149.126
C09799=1145.067,38.308,-50.473,-179.918,6.338,149.126
C09800=1145.072,38.058,-50.457,-179.920,6.338,149.127
C09801=1145.076,37.808,-50.443,-179.924,6.336,149.128
C09802=1145.082,37.559,-50.427,-179.926,6.335,149.128
C09803=1145.087,37.309,-50.413,-179.929,6.335,149.129
C09804=1145.091,37.060,-50.398,-179.931,6.333,149.129
C09805=1145.097,36.810,-50.383,-179.933,6.333,149.130
C09806=1145.102,36.561,-50.368,-179.937,6.331,149.130
C09807=1145.107,36.311,-50.352,-179.939,6.330,149.131
C09808=1145.112,36.062,-50.338,-179.942,6.329,149.131
C09809=1145.117,35.813,-50.323,-179.944,6.328,149.132
C09810=1145.122,35.563,-50.308,-179.946,6.328,149.132
C09811=1145.127,35.314,-50.293,-179.950,6.326,149.133
C09812=1145.132,35.064,-50.279,-179.952,6.325,149.133
C09813=1145.137,34.814,-50.263,-179.955,6.324,149.134
C09814=1145.142,34.565,-50.249,-179.957,6.323,149.134
C09815=1145.147,34.316,-50.234,-179.959,6.323,149.135
C09816=1145.153,34.066,-50.219,-179.963,6.321,149.136
C09817=1145.157,33.817,-50.204,-179.965,6.320,149.136
C09818=1145.162,33.567,-50.190,-179.968,6.319,149.137
C09819=1145.168,33.317,-50.174,-179.970,6.318,149.137
C09820=1145.173,33.068,-50.160,-179.972,6.317,149.138
C09821=1145.178,32.818,-50.146,-179.976,6.316,149.138
C09822=1145.183,32.569,-50.130,-179.978,6.315,149.139
C09823=1145.188,32.319,-50.116,-179.980,6.315,149.139
C09824=1145.193,32.070,-50.101,-179.983,6.313,149.140
C09825=1145.198,31.820,-50.087,-179.985,6.312,149.140
C09826=1145.204,31.571,-50.072,-179.989,6.311,149.141
C09827=1145.209,31.322,-50.057,-179.991,6.310,149.141
C09828=1145.214,31.072,-50.043,-179.993,6.310,149.142
C09829=1145.218,30.823,-50.028,-179.996,6.308,149.143
C09830=1145.224,30.573,-50.013,-179.998,6.307,149.143
C09831=1145.229,30.323,-49.999,179.998,6.306,149.144
C09832=1145.233,30.074,-49.984,179.996,6.305,149.144
C09833=1145.238,29.824,-49.969,179.994,6.305,149.145
C09834=1145.243,29.575,-49.955,179.991,6.303,149.145
C09835=1145.249,29.325,-49.940,179.989,6.302,149.146
C09836=1145.254,29.075,-49.925,179.986,6.302,149.146
C09837=1145.259,28.826,-49.911,179.983,6.300,149.147
C09838=1145.264,28.576,-49.897,179.981,6.300,149.148
C09839=1145.269,28.328,-49.882,179.978,6.299,149.148
C09840=1145.275,28.078,-49.867,179.976,6.297,149.148
C09841=1145.280,27.809,-49.852,179.973,6.297,149.149
C09842=1145.285,27.539,-49.837,179.970,6.296,149.150
C09843=1145.290,27.271,-49.821,179.968,6.295,149.150
C09844=1145.296,27.002,-49.805,179.964,6.294,149.151
C09845=1145.301,26.752,-49.790,179.962,6.293,149.151
C09846=1145.306,26.502,-49.776,179.959,6.292,149.152
C09847=1145.312,26.253,-49.762,179.957,6.291,149.153
C09848=1145.317,26.003,-49.748,179.955,6.290,149.153
C09849=1145.321,25.754,-49.733,179.951,6.289,149.154
C09850=1145.326,25.505,-49.718,179.949,6.288,149.154
C09851=1145.331,25.255,-49.704,179.947,6.287,149.155
C09852=1145.336,25.005,-49.690,179.944,6.286,149.155
C09853=1145.342,24.756,-49.675,179.941,6.285,149.156
C09854=1145.347,24.506,-49.661,179.939,6.285,149.156
C09855=1145.352,24.256,-49.647,179.936,6.283,149.157
C09856=1145.357,24.007,-49.632,179.934,6.282,149.158
C09857=1145.362,23.758,-49.618,179.931,6.282,149.158
C09858=1145.367,23.508,-49.603,179.928,6.280,149.159
C09859=1145.372,23.259,-49.589,179.926,6.280,149.159
C09860=1145.377,23.009,-49.575,179.924,6.279,149.160
C09861=1145.382,22.760,-49.561,179.921,6.277,149.160
C09862=1145.387,22.510,-49.547,179.918,6.277,149.161
C09863=1145.392,22.260,-49.532,179.916,6.276,149.161
C09864=1145.398,22.011,-49.518,179.913,6.275,149.162
C09865=1145.403,21.761,-49.504,179.911,6.274,149.162
C09866=1145.408,21.512,-49.490,179.908,6.273,149.163
C09867=1145.413,21.262,-49.476,179.906,6.272,149.163
C09868=1145.418,21.013,-49.462,179.903,6.271,149.164
C09869=1145.423,20.763,-49.447,179.901,6.270,149.165
C09870=1145.428,20.514,-49.433,179.898,6.270,149.165
C09871=1145.433,20.264,-49.419,179.895,6.268,149.166
C09872=1145.439,20.015,-49.405,179.893,6.268,149.166
C09873=1145.444,19.765,-49.391,179.890,6.267,149.167
C09874=1145.448,19.515,-49.376,179.888,6.265,149.167
C09875=1145.453,19.266,-49.362,179.885,6.265,149.168
C09876=1145.459,19.017,-49.348,179.883,6.264,149.168
C09877=1145.464,18.767,-49.334,179.880,6.264,149.169
C09878=1145.469,18.517,-49.320,179.877,6.262,149.170
C09879=1145.473,18.268,-49.306,179.875,6.261,149.170
C09880=1145.479,18.018,-49.293,179.873,6.261,149.171
C09881=1145.484,17.769,-49.278,179.870,6.259,149.171
C09882=1145.489,17.519,-49.264,179.867,6.259,149.172
C09883=1145.494,17.270,-49.250,179.865,6.258,149.172
C09884=1145.499,17.020,-49.236,179.863,6.257,149.173
C09885=1145.504,16.770,-49.222,179.860,6.256,149.174
C09886=1145.509,16.521,-49.207,179.857,6.255,149.174
C09887=1145.515,16.271,-49.194,179.855,6.255,149.175
C09888=1145.519,16.022,-49.181,179.852,6.253,149.175
C09889=1145.524,15.772,-49.166,179.849,6.253,149.176
C09890=1145.530,15.523,-49.152,179.847,6.252,149.176
C09891=1145.535,15.273,-49.138,179.845,6.251,149.177
C09892=1145.540,15.023,-49.125,179.842,6.250,149.177
C09893=1145.546,14.774,-49.111,179.840,6.249,149.178
C09894=1145.550,14.524,-49.097,179.837,6.248,149.179
C09895=1145.555,14.275,-49.083,179.835,6.248,149.179
C09896=1145.561,14.025,-49.069,179.831,6.246,149.180
C09897=1145.566,13.775,-49.055,179.829,6.246,149.180
C09898=1145.571,13.526,-49.041,179.827,6.245,149.181
C09899=1145.575,13.277,-49.028,179.824,6.243,149.181
C09900=1145.581,13.027,-49.014,179.822,6.243,149.182
C09901=1145.586,12.778,-49.000,179.819,6.242,149.182
C09902=1145.591,12.528,-48.986,179.817,6.241,149.183
C09903=1145.596,12.278,-48.972,179.814,6.240,149.184
C09904=1145.601,12.029,-48.959,179.811,6.239,149.184
C09905=1145.606,11.779,-48.945,179.809,6.239,149.184
C09906=1145.612,11.530,-48.932,179.807,6.238,149.185
C09907=1145.617,11.280,-48.917,179.804,6.236,149.186
C09908=1145.621,11.030,-48.904,179.801,6.236,149.186
C09909=1145.627,10.781,-48.890,179.799,6.235,149.187
C09910=1145.632,10.531,-48.876,179.797,6.234,149.187
C09911=1145.638,10.282,-48.862,179.794,6.234,149.188
C09912=1145.642,10.032,-48.849,179.791,6.232,149.188
C09913=1145.647,9.782,-48.835,179.789,6.232,149.189
C09914=1145.653,9.533,-48.822,179.787,6.231,149.190
C09915=1145.657,9.283,-48.808,179.784,6.231,149.190
C09916=1145.663,9.034,-48.795,179.781,6.229,149.191
C09917=1145.668,8.784,-48.781,179.779,6.228,149.191
C09918=1145.673,8.535,-48.767,179.776,6.228,149.192
C09919=1145.678,8.285,-48.754,179.774,6.227,149.192
C09920=1145.683,8.035,-48.739,179.771,6.226,149.193
C09921=1145.688,7.786,-48.727,179.769,6.225,149.193
C09922=1145.693,7.536,-48.713,179.766,6.224,149.194
C09923=1145.699,7.287,-48.699,179.764,6.224,149.195
C09924=1145.703,7.037,-48.686,179.762,6.223,149.195
C09925=1145.709,6.788,-48.672,179.759,6.222,149.196
C09926=1145.714,6.538,-48.658,179.756,6.221,149.196
C09927=1145.719,6.289,-48.646,179.754,6.220,149.197
C09928=1145.724,6.039,-48.631,179.752,6.220,149.197
C09929=1145.729,5.790,-48.619,179.749,6.219,149.198
C09930=1145.734,5.540,-48.604,179.746,6.217,149.198
C09931=1145.740,5.290,-48.591,179.743,6.217,149.199
C09932=1145.745,5.040,-48.578,179.741,6.216,149.200
C09933=1145.750,4.791,-48.564,179.739,6.215,149.200
C09934=1145.755,4.541,-48.551,179.736,6.215,149.201
C09935=1145.760,4.292,-48.537,179.734,6.213,149.201
C09936=1145.765,4.042,-48.525,179.731,6.213,149.202
C09937=1145.771,3.793,-48.511,179.729,6.212,149.202
C09938=1145.776,3.543,-48.497,179.726,6.212,149.203
C09939=1145.781,3.293,-48.484,179.724,6.211,149.204
C09940=1145.786,3.044,-48.470,179.721,6.209,149.204
C09941=1145.791,2.794,-48.458,179.719,6.209,149.205
C09942=1145.796,2.544,-48.444,179.716,6.208,149.205
C09943=1145.801,2.295,-48.431,179.714,6.208,149.206
C09944=1145.806,2.045,-48.417,179.712,6.207,149.206
C09945=1145.812,1.776,-48.404,179.708,6.206,149.207
C09946=1145.817,1.507,-48.389,179.706,6.205,149.207
C09947=1145.823,1.237,-48.375,179.703,6.204,149.208
C09948=1145.829,0.968,-48.360,179.700,6.203,149.209
C09949=1145.833,0.718,-48.347,179.698,6.202,149.209
C09950=1145.839,0.468,-48.334,179.696,6.201,149.210
C09951=1145.843,0.219,-48.320,179.693,6.201,149.210
C09952=1145.849,-0.030,-48.307,179.690,6.199,149.211
C09953=1145.854,-0.281,-48.294,179.688,6.199,149.212
C09954=1145.859,-0.530,-48.281,179.686,6.198,149.212
C09955=1145.865,-0.779,-48.267,179.683,6.198,149.213
C09956=1145.869,-1.029,-48.254,179.681,6.197,149.213
C09957=1145.875,-1.279,-48.241,179.679,6.196,149.214
C09958=1145.879,-1.529,-48.228,179.675,6.195,149.214
C09959=1145.885,-1.778,-48.215,179.673,6.194,149.215
C09960=1145.890,-2.027,-48.202,179.671,6.194,149.216
C09961=1145.895,-2.277,-48.189,179.668,6.193,149.216
C09962=1145.901,-2.527,-48.176,179.666,6.192,149.217
C09963=1145.906,-2.776,-48.163,179.664,6.192,149.217
C09964=1145.911,-3.026,-48.149,179.661,6.191,149.218
C09965=1145.916,-3.276,-48.137,179.658,6.190,149.218
C09966=1145.921,-3.524,-48.124,179.656,6.189,149.219
C09967=1145.926,-3.775,-48.110,179.653,6.188,149.219
C09968=1145.931,-4.024,-48.097,179.651,6.187,149.220
C09969=1145.937,-4.274,-48.084,179.648,6.187,149.221
C09970=1145.942,-4.524,-48.071,179.646,6.186,149.221
C09971=1145.947,-4.773,-48.059,179.644,6.186,149.222
C09972=1145.952,-5.023,-48.045,179.641,6.184,149.222
C09973=1145.957,-5.273,-48.032,179.639,6.183,149.223
C09974=1145.962,-5.522,-48.020,179.636,6.183,149.223
C09975=1145.968,-5.772,-48.006,179.634,6.182,149.224
C09976=1145.973,-6.022,-47.994,179.631,6.182,149.225
C09977=1145.977,-6.270,-47.980,179.629,6.181,149.225
C09978=1145.983,-6.521,-47.967,179.626,6.180,149.226
C09979=1145.988,-6.770,-47.954,179.624,6.179,149.226
C09980=1145.993,-7.019,-47.942,179.621,6.178,149.227
C09981=1145.998,-7.269,-47.929,179.619,6.178,149.227
C09982=1146.003,-7.519,-47.915,179.617,6.177,149.228
C09983=1146.008,-7.768,-47.903,179.614,6.176,149.229
C09984=1146.014,-8.018,-47.890,179.612,6.176,149.229
C09985=1146.019,-8.268,-47.877,179.609,6.175,149.230
C09986=1146.024,-8.517,-47.864,179.607,6.174,149.230
C09987=1146.029,-8.767,-47.851,179.604,6.173,149.231
C09988=1146.035,-9.016,-47.840,179.601,6.172,149.231
C09989=1146.039,-9.267,-47.827,179.599,6.172,149.232
C09990=1146.045,-9.516,-47.813,179.597,6.171,149.232
C09991=1146.050,-9.765,-47.801,179.594,6.170,149.233
C09992=1146.055,-10.015,-47.788,179.592,6.170,149.234
C09993=1146.060,-10.265,-47.775,179.590,6.169,149.234
C09994=1146.066,-10.514,-47.762,179.587,6.168,149.235
C09995=1146.071,-10.764,-47.749,179.585,6.168,149.235
C09996=1146.075,-11.014,-47.736,179.582,6.166,149.236
//INST
///DATE 2021/06/15 17:27
///ATTR SC,RW,RJ
////FRAME ROBOT
///GROUP1 RB1
NOP
MOVL C00000 V=800.0 PL=0
MOVL C00001 V=800.0 PL=0
MOVL C00002 V=800.0 PL=0
MOVL C00003 V=800.0 PL=0
MOVL C00004 V=800.0 PL=0
MOVL C00005 V=800.0 PL=0
MOVL C00006 V=800.0 PL=0
MOVL C00007 V=800.0 PL=0
MOVL C00008 V=800.0 PL=0
MOVL C00009 V=800.0 PL=0
MOVL C00010 V=800.0 PL=0
MOVL C00011 V=800.0 PL=0
MOVL C00012 V=800.0 PL=0
MOVL C00013 V=800.0 PL=0
MOVL C00014 V=800.0 PL=0
MOVL C00015 V=800.0 PL=0
MOVL C00016 V=800.0 PL=0
MOVL C00017 V=800.0 PL=0
MOVL C00018 V=800.0 PL=0
MOVL C00019 V=800.0 PL=0
MOVL C00020 V=800.0 PL=0
MOVL C00021 V=800.0 PL=0
MOVL C00022 V=800.0 PL=0
MOVL C00023 V=800.0 PL=0
MOVL C00024 V=800.0 PL=0
MOVL C00025 V=800.0 PL=0
MOVL C00026 V=800.0 PL=0
MOVL C00027 V=800.0 PL=0
MOVL C00028 V=800.0 PL=0
MOVL C00029 V=800.0 PL=0
MOVL C00030 V=800.0 PL=0
MOVL C00031 V=800.0 PL=0
MOVL C00032 V=800.0 PL=0
MOVL C00033 V=800.0 PL=0
MOVL C00034 V=800.0 PL=0
MOVL C00035 V=800.0 PL=0
MOVL C00036 V=800.0 PL=0
MOVL C00037 V=800.0 PL=0
MOVL C00038 V=800.0 PL=0
MOVL C00039 V=800.0 PL=0
MOVL C00040 V=800.0 PL=0
MOVL C00041 V=800.0 PL=0
MOVL C00042 V=800.0 PL=0
MOVL C00043 V=800.0 PL=0
MOVL C00044 V=800.0 PL=0
MOVL C00045 V=800.0 PL=0
MOVL C00046 V=800.0 PL=0
MOVL C00047 V=800.0 PL=0
MOVL C00048 V=800.0 PL=0
MOVL C00049 V=800.0 PL=0
MOVL C00050 V=800.0 PL=0
MOVL C00051 V=800.0 PL=0
MOVL C00052 V=800.0 PL=0
MOVL C00053 V=800.0 PL=0
MOVL C00054 V=800.0 PL=0
MOVL C00055 V=800.0 PL=0
MOVL C00056 V=800.0 PL=0
MOVL C00057 V=800.0 PL=0
MOVL C00058 V=800.0 PL=0
MOVL C00059 V=800.0 PL=0
MOVL C00060 V=800.0 PL=0
MOVL C00061 V=800.0 PL=0
MOVL C00062 V=800.0 PL=0
MOVL C00063 V=800.0 PL=0
MOVL C00064 V=800.0 PL=0
MOVL C00065 V=800.0 PL=0
MOVL C00066 V=800.0 PL=0
MOVL C00067 V=800.0 PL=0
MOVL C00068 V=800.0 PL=0
MOVL C00069 V=800.0 PL=0
MOVL C00070 V=800.0 PL=0
MOVL C00071 V=800.0 PL=0
MOVL C00072 V=800.0 PL=0
MOVL C00073 V=800.0 PL=0
MOVL C00074 V=800.0 PL=0
MOVL C00075 V=800.0 PL=0
MOVL C00076 V=800.0 PL=0
MOVL C00077 V=800.0 PL=0
MOVL C00078 V=800.0 PL=0
MOVL C00079 V=800.0 PL=0
MOVL C00080 V=800.0 PL=0
MOVL C00081 V=800.0 PL=0
MOVL C00082 V=800.0 PL=0
MOVL C00083 V=800.0 PL=0
MOVL C00084 V=800.0 PL=0
MOVL C00085 V=800.0 PL=0
MOVL C00086 V=800.0 PL=0
MOVL C00087 V=800.0 PL=0
MOVL C00088 V=800.0 PL=0
MOVL C00089 V=800.0 PL=0
MOVL C00090 V=800.0 PL=0
MOVL C00091 V=800.0 PL=0
MOVL C00092 V=800.0 PL=0
MOVL C00093 V=800.0 PL=0
MOVL C00094 V=800.0 PL=0
MOVL C00095 V=800.0 PL=0
MOVL C00096 V=800.0 PL=0
MOVL C00097 V=800.0 PL=0
MOVL C00098 V=800.0 PL=0
MOVL C00099 V=800.0 PL=0
MOVL C00100 V=800.0 PL=0
MOVL C00101 V=800.0 PL=0
MOVL C00102 V=800.0 PL=0
MOVL C00103 V=800.0 PL=0
MOVL C00104 V=800.0 PL=0
MOVL C00105 V=800.0 PL=0
MOVL C00106 V=800.0 PL=0
MOVL C00107 V=800.0 PL=0
MOVL C00108 V=800.0 PL=0
MOVL C00109 V=800.0 PL=0
MOVL C00110 V=800.0 PL=0
MOVL C00111 V=800.0 PL=0
MOVL C00112 V=800.0 PL=0
MOVL C00113 V=800.0 PL=0
MOVL C00114 V=800.0 PL=0
MOVL C00115 V=800.0 PL=0
MOVL C00116 V=800.0 PL=0
MOVL C00117 V=800.0 PL=0
MOVL C00118 V=800.0 PL=0
MOVL C00119 V=800.0 PL=0
MOVL C00120 V=800.0 PL=0
MOVL C00121 V=800.0 PL=0
MOVL C00122 V=800.0 PL=0
MOVL C00123 V=800.0 PL=0
MOVL C00124 V=800.0 PL=0
MOVL C00125 V=800.0 PL=0
MOVL C00126 V=800.0 PL=0
MOVL C00127 V=800.0 PL=0
MOVL C00128 V=800.0 PL=0
MOVL C00129 V=800.0 PL=0
MOVL C00130 V=800.0 PL=0
MOVL C00131 V=800.0 PL=0
MOVL C00132 V=800.0 PL=0
MOVL C00133 V=800.0 PL=0
MOVL C00134 V=800.0 PL=0
MOVL C00135 V=800.0 PL=0
MOVL C00136 V=800.0 PL=0
MOVL C00137 V=800.0 PL=0
MOVL C00138 V=800.0 PL=0
MOVL C00139 V=800.0 PL=0
MOVL C00140 V=800.0 PL=0
MOVL C00141 V=800.0 PL=0
MOVL C00142 V=800.0 PL=0
MOVL C00143 V=800.0 PL=0
MOVL C00144 V=800.0 PL=0
MOVL C00145 V=800.0 PL=0
MOVL C00146 V=800.0 PL=0
MOVL C00147 V=800.0 PL=0
MOVL C00148 V=800.0 PL=0
MOVL C00149 V=800.0 PL=0
MOVL C00150 V=800.0 PL=0
MOVL C00151 V=800.0 PL=0
MOVL C00152 V=800.0 PL=0
MOVL C00153 V=800.0 PL=0
MOVL C00154 V=800.0 PL=0
MOVL C00155 V=800.0 PL=0
MOVL C00156 V=800.0 PL=0
MOVL C00157 V=800.0 PL=0
MOVL C00158 V=800.0 PL=0
MOVL C00159 V=800.0 PL=0
MOVL C00160 V=800.0 PL=0
MOVL C00161 V=800.0 PL=0
MOVL C00162 V=800.0 PL=0
MOVL C00163 V=800.0 PL=0
MOVL C00164 V=800.0 PL=0
MOVL C00165 V=800.0 PL=0
MOVL C00166 V=800.0 PL=0
MOVL C00167 V=800.0 PL=0
MOVL C00168 V=800.0 PL=0
MOVL C00169 V=800.0 PL=0
MOVL C00170 V=800.0 PL=0
MOVL C00171 V=800.0 PL=0
MOVL C00172 V=800.0 PL=0
MOVL C00173 V=800.0 PL=0
MOVL C00174 V=800.0 PL=0
MOVL C00175 V=800.0 PL=0
MOVL C00176 V=800.0 PL=0
MOVL C00177 V=800.0 PL=0
MOVL C00178 V=800.0 PL=0
MOVL C00179 V=800.0 PL=0
MOVL C00180 V=800.0 PL=0
MOVL C00181 V=800.0 PL=0
MOVL C00182 V=800.0 PL=0
MOVL C00183 V=800.0 PL=0
MOVL C00184 V=800.0 PL=0
MOVL C00185 V=800.0 PL=0
MOVL C00186 V=800.0 PL=0
MOVL C00187 V=800.0 PL=0
MOVL C00188 V=800.0 PL=0
MOVL C00189 V=800.0 PL=0
MOVL C00190 V=800.0 PL=0
MOVL C00191 V=800.0 PL=0
MOVL C00192 V=800.0 PL=0
MOVL C00193 V=800.0 PL=0
MOVL C00194 V=800.0 PL=0
MOVL C00195 V=800.0 PL=0
MOVL C00196 V=800.0 PL=0
MOVL C00197 V=800.0 PL=0
MOVL C00198 V=800.0 PL=0
MOVL C00199 V=800.0 PL=0
MOVL C00200 V=800.0 PL=0
MOVL C00201 V=800.0 PL=0
MOVL C00202 V=800.0 PL=0
MOVL C00203 V=800.0 PL=0
MOVL C00204 V=800.0 PL=0
MOVL C00205 V=800.0 PL=0
MOVL C00206 V=800.0 PL=0
MOVL C00207 V=800.0 PL=0
MOVL C00208 V=800.0 PL=0
MOVL C00209 V=800.0 PL=0
MOVL C00210 V=800.0 PL=0
MOVL C00211 V=800.0 PL=0
MOVL C00212 V=800.0 PL=0
MOVL C00213 V=800.0 PL=0
MOVL C00214 V=800.0 PL=0
MOVL C00215 V=800.0 PL=0
MOVL C00216 V=800.0 PL=0
MOVL C00217 V=800.0 PL=0
MOVL C00218 V=800.0 PL=0
MOVL C00219 V=800.0 PL=0
MOVL C00220 V=800.0 PL=0
MOVL C00221 V=800.0 PL=0
MOVL C00222 V=800.0 PL=0
MOVL C00223 V=800.0 PL=0
MOVL C00224 V=800.0 PL=0
MOVL C00225 V=800.0 PL=0
MOVL C00226 V=800.0 PL=0
MOVL C00227 V=800.0 PL=0
MOVL C00228 V=800.0 PL=0
MOVL C00229 V=800.0 PL=0
MOVL C00230 V=800.0 PL=0
MOVL C00231 V=800.0 PL=0
MOVL C00232 V=800.0 PL=0
MOVL C00233 V=800.0 PL=0
MOVL C00234 V=800.0 PL=0
MOVL C00235 V=800.0 PL=0
MOVL C00236 V=800.0 PL=0
MOVL C00237 V=800.0 PL=0
MOVL C00238 V=800.0 PL=0
MOVL C00239 V=800.0 PL=0
MOVL C00240 V=800.0 PL=0
MOVL C00241 V=800.0 PL=0
MOVL C00242 V=800.0 PL=0
MOVL C00243 V=800.0 PL=0
MOVL C00244 V=800.0 PL=0
MOVL C00245 V=800.0 PL=0
MOVL C00246 V=800.0 PL=0
MOVL C00247 V=800.0 PL=0
MOVL C00248 V=800.0 PL=0
MOVL C00249 V=800.0 PL=0
MOVL C00250 V=800.0 PL=0
MOVL C00251 V=800.0 PL=0
MOVL C00252 V=800.0 PL=0
MOVL C00253 V=800.0 PL=0
MOVL C00254 V=800.0 PL=0
MOVL C00255 V=800.0 PL=0
MOVL C00256 V=800.0 PL=0
MOVL C00257 V=800.0 PL=0
MOVL C00258 V=800.0 PL=0
MOVL C00259 V=800.0 PL=0
MOVL C00260 V=800.0 PL=0
MOVL C00261 V=800.0 PL=0
MOVL C00262 V=800.0 PL=0
MOVL C00263 V=800.0 PL=0
MOVL C00264 V=800.0 PL=0
MOVL C00265 V=800.0 PL=0
MOVL C00266 V=800.0 PL=0
MOVL C00267 V=800.0 PL=0
MOVL C00268 V=800.0 PL=0
MOVL C00269 V=800.0 PL=0
MOVL C00270 V=800.0 PL=0
MOVL C00271 V=800.0 PL=0
MOVL C00272 V=800.0 PL=0
MOVL C00273 V=800.0 PL=0
MOVL C00274 V=800.0 PL=0
MOVL C00275 V=800.0 PL=0
MOVL C00276 V=800.0 PL=0
MOVL C00277 V=800.0 PL=0
MOVL C00278 V=800.0 PL=0
MOVL C00279 V=800.0 PL=0
MOVL C00280 V=800.0 PL=0
MOVL C00281 V=800.0 PL=0
MOVL C00282 V=800.0 PL=0
MOVL C00283 V=800.0 PL=0
MOVL C00284 V=800.0 PL=0
MOVL C00285 V=800.0 PL=0
MOVL C00286 V=800.0 PL=0
MOVL C00287 V=800.0 PL=0
MOVL C00288 V=800.0 PL=0
MOVL C00289 V=800.0 PL=0
MOVL C00290 V=800.0 PL=0
MOVL C00291 V=800.0 PL=0
MOVL C00292 V=800.0 PL=0
MOVL C00293 V=800.0 PL=0
MOVL C00294 V=800.0 PL=0
MOVL C00295 V=800.0 PL=0
MOVL C00296 V=800.0 PL=0
MOVL C00297 V=800.0 PL=0
MOVL C00298 V=800.0 PL=0
MOVL C00299 V=800.0 PL=0
MOVL C00300 V=800.0 PL=0
MOVL C00301 V=800.0 PL=0
MOVL C00302 V=800.0 PL=0
MOVL C00303 V=800.0 PL=0
MOVL C00304 V=800.0 PL=0
MOVL C00305 V=800.0 PL=0
MOVL C00306 V=800.0 PL=0
MOVL C00307 V=800.0 PL=0
MOVL C00308 V=800.0 PL=0
MOVL C00309 V=800.0 PL=0
MOVL C00310 V=800.0 PL=0
MOVL C00311 V=800.0 PL=0
MOVL C00312 V=800.0 PL=0
MOVL C00313 V=800.0 PL=0
MOVL C00314 V=800.0 PL=0
MOVL C00315 V=800.0 PL=0
MOVL C00316 V=800.0 PL=0
MOVL C00317 V=800.0 PL=0
MOVL C00318 V=800.0 PL=0
MOVL C00319 V=800.0 PL=0
MOVL C00320 V=800.0 PL=0
MOVL C00321 V=800.0 PL=0
MOVL C00322 V=800.0 PL=0
MOVL C00323 V=800.0 PL=0
MOVL C00324 V=800.0 PL=0
MOVL C00325 V=800.0 PL=0
MOVL C00326 V=800.0 PL=0
MOVL C00327 V=800.0 PL=0
MOVL C00328 V=800.0 PL=0
MOVL C00329 V=800.0 PL=0
MOVL C00330 V=800.0 PL=0
MOVL C00331 V=800.0 PL=0
MOVL C00332 V=800.0 PL=0
MOVL C00333 V=800.0 PL=0
MOVL C00334 V=800.0 PL=0
MOVL C00335 V=800.0 PL=0
MOVL C00336 V=800.0 PL=0
MOVL C00337 V=800.0 PL=0
MOVL C00338 V=800.0 PL=0
MOVL C00339 V=800.0 PL=0
MOVL C00340 V=800.0 PL=0
MOVL C00341 V=800.0 PL=0
MOVL C00342 V=800.0 PL=0
MOVL C00343 V=800.0 PL=0
MOVL C00344 V=800.0 PL=0
MOVL C00345 V=800.0 PL=0
MOVL C00346 V=800.0 PL=0
MOVL C00347 V=800.0 PL=0
MOVL C00348 V=800.0 PL=0
MOVL C00349 V=800.0 PL=0
MOVL C00350 V=800.0 PL=0
MOVL C00351 V=800.0 PL=0
MOVL C00352 V=800.0 PL=0
MOVL C00353 V=800.0 PL=0
MOVL C00354 V=800.0 PL=0
MOVL C00355 V=800.0 PL=0
MOVL C00356 V=800.0 PL=0
MOVL C00357 V=800.0 PL=0
MOVL C00358 V=800.0 PL=0
MOVL C00359 V=800.0 PL=0
MOVL C00360 V=800.0 PL=0
MOVL C00361 V=800.0 PL=0
MOVL C00362 V=800.0 PL=0
MOVL C00363 V=800.0 PL=0
MOVL C00364 V=800.0 PL=0
MOVL C00365 V=800.0 PL=0
MOVL C00366 V=800.0 PL=0
MOVL C00367 V=800.0 PL=0
MOVL C00368 V=800.0 PL=0
MOVL C00369 V=800.0 PL=0
MOVL C00370 V=800.0 PL=0
MOVL C00371 V=800.0 PL=0
MOVL C00372 V=800.0 PL=0
MOVL C00373 V=800.0 PL=0
MOVL C00374 V=800.0 PL=0
MOVL C00375 V=800.0 PL=0
MOVL C00376 V=800.0 PL=0
MOVL C00377 V=800.0 PL=0
MOVL C00378 V=800.0 PL=0
MOVL C00379 V=800.0 PL=0
MOVL C00380 V=800.0 PL=0
MOVL C00381 V=800.0 PL=0
MOVL C00382 V=800.0 PL=0
MOVL C00383 V=800.0 PL=0
MOVL C00384 V=800.0 PL=0
MOVL C00385 V=800.0 PL=0
MOVL C00386 V=800.0 PL=0
MOVL C00387 V=800.0 PL=0
MOVL C00388 V=800.0 PL=0
MOVL C00389 V=800.0 PL=0
MOVL C00390 V=800.0 PL=0
MOVL C00391 V=800.0 PL=0
MOVL C00392 V=800.0 PL=0
MOVL C00393 V=800.0 PL=0
MOVL C00394 V=800.0 PL=0
MOVL C00395 V=800.0 PL=0
MOVL C00396 V=800.0 PL=0
MOVL C00397 V=800.0 PL=0
MOVL C00398 V=800.0 PL=0
MOVL C00399 V=800.0 PL=0
MOVL C00400 V=800.0 PL=0
MOVL C00401 V=800.0 PL=0
MOVL C00402 V=800.0 PL=0
MOVL C00403 V=800.0 PL=0
MOVL C00404 V=800.0 PL=0
MOVL C00405 V=800.0 PL=0
MOVL C00406 V=800.0 PL=0
MOVL C00407 V=800.0 PL=0
MOVL C00408 V=800.0 PL=0
MOVL C00409 V=800.0 PL=0
MOVL C00410 V=800.0 PL=0
MOVL C00411 V=800.0 PL=0
MOVL C00412 V=800.0 PL=0
MOVL C00413 V=800.0 PL=0
MOVL C00414 V=800.0 PL=0
MOVL C00415 V=800.0 PL=0
MOVL C00416 V=800.0 PL=0
MOVL C00417 V=800.0 PL=0
MOVL C00418 V=800.0 PL=0
MOVL C00419 V=800.0 PL=0
MOVL C00420 V=800.0 PL=0
MOVL C00421 V=800.0 PL=0
MOVL C00422 V=800.0 PL=0
MOVL C00423 V=800.0 PL=0
MOVL C00424 V=800.0 PL=0
MOVL C00425 V=800.0 PL=0
MOVL C00426 V=800.0 PL=0
MOVL C00427 V=800.0 PL=0
MOVL C00428 V=800.0 PL=0
MOVL C00429 V=800.0 PL=0
MOVL C00430 V=800.0 PL=0
MOVL C00431 V=800.0 PL=0
MOVL C00432 V=800.0 PL=0
MOVL C00433 V=800.0 PL=0
MOVL C00434 V=800.0 PL=0
MOVL C00435 V=800.0 PL=0
MOVL C00436 V=800.0 PL=0
MOVL C00437 V=800.0 PL=0
MOVL C00438 V=800.0 PL=0
MOVL C00439 V=800.0 PL=0
MOVL C00440 V=800.0 PL=0
MOVL C00441 V=800.0 PL=0
MOVL C00442 V=800.0 PL=0
MOVL C00443 V=800.0 PL=0
MOVL C00444 V=800.0 PL=0
MOVL C00445 V=800.0 PL=0
MOVL C00446 V=800.0 PL=0
MOVL C00447 V=800.0 PL=0
MOVL C00448 V=800.0 PL=0
MOVL C00449 V=800.0 PL=0
MOVL C00450 V=800.0 PL=0
MOVL C00451 V=800.0 PL=0
MOVL C00452 V=800.0 PL=0
MOVL C00453 V=800.0 PL=0
MOVL C00454 V=800.0 PL=0
MOVL C00455 V=800.0 PL=0
MOVL C00456 V=800.0 PL=0
MOVL C00457 V=800.0 PL=0
MOVL C00458 V=800.0 PL=0
MOVL C00459 V=800.0 PL=0
MOVL C00460 V=800.0 PL=0
MOVL C00461 V=800.0 PL=0
MOVL C00462 V=800.0 PL=0
MOVL C00463 V=800.0 PL=0
MOVL C00464 V=800.0 PL=0
MOVL C00465 V=800.0 PL=0
MOVL C00466 V=800.0 PL=0
MOVL C00467 V=800.0 PL=0
MOVL C00468 V=800.0 PL=0
MOVL C00469 V=800.0 PL=0
MOVL C00470 V=800.0 PL=0
MOVL C00471 V=800.0 PL=0
MOVL C00472 V=800.0 PL=0
MOVL C00473 V=800.0 PL=0
MOVL C00474 V=800.0 PL=0
MOVL C00475 V=800.0 PL=0
MOVL C00476 V=800.0 PL=0
MOVL C00477 V=800.0 PL=0
MOVL C00478 V=800.0 PL=0
MOVL C00479 V=800.0 PL=0
MOVL C00480 V=800.0 PL=0
MOVL C00481 V=800.0 PL=0
MOVL C00482 V=800.0 PL=0
MOVL C00483 V=800.0 PL=0
MOVL C00484 V=800.0 PL=0
MOVL C00485 V=800.0 PL=0
MOVL C00486 V=800.0 PL=0
MOVL C00487 V=800.0 PL=0
MOVL C00488 V=800.0 PL=0
MOVL C00489 V=800.0 PL=0
MOVL C00490 V=800.0 PL=0
MOVL C00491 V=800.0 PL=0
MOVL C00492 V=800.0 PL=0
MOVL C00493 V=800.0 PL=0
MOVL C00494 V=800.0 PL=0
MOVL C00495 V=800.0 PL=0
MOVL C00496 V=800.0 PL=0
MOVL C00497 V=800.0 PL=0
MOVL C00498 V=800.0 PL=0
MOVL C00499 V=800.0 PL=0
MOVL C00500 V=800.0 PL=0
MOVL C00501 V=800.0 PL=0
MOVL C00502 V=800.0 PL=0
MOVL C00503 V=800.0 PL=0
MOVL C00504 V=800.0 PL=0
MOVL C00505 V=800.0 PL=0
MOVL C00506 V=800.0 PL=0
MOVL C00507 V=800.0 PL=0
MOVL C00508 V=800.0 PL=0
MOVL C00509 V=800.0 PL=0
MOVL C00510 V=800.0 PL=0
MOVL C00511 V=800.0 PL=0
MOVL C00512 V=800.0 PL=0
MOVL C00513 V=800.0 PL=0
MOVL C00514 V=800.0 PL=0
MOVL C00515 V=800.0 PL=0
MOVL C00516 V=800.0 PL=0
MOVL C00517 V=800.0 PL=0
MOVL C00518 V=800.0 PL=0
MOVL C00519 V=800.0 PL=0
MOVL C00520 V=800.0 PL=0
MOVL C00521 V=800.0 PL=0
MOVL C00522 V=800.0 PL=0
MOVL C00523 V=800.0 PL=0
MOVL C00524 V=800.0 PL=0
MOVL C00525 V=800.0 PL=0
MOVL C00526 V=800.0 PL=0
MOVL C00527 V=800.0 PL=0
MOVL C00528 V=800.0 PL=0
MOVL C00529 V=800.0 PL=0
MOVL C00530 V=800.0 PL=0
MOVL C00531 V=800.0 PL=0
MOVL C00532 V=800.0 PL=0
MOVL C00533 V=800.0 PL=0
MOVL C00534 V=800.0 PL=0
MOVL C00535 V=800.0 PL=0
MOVL C00536 V=800.0 PL=0
MOVL C00537 V=800.0 PL=0
MOVL C00538 V=800.0 PL=0
MOVL C00539 V=800.0 PL=0
MOVL C00540 V=800.0 PL=0
MOVL C00541 V=800.0 PL=0
MOVL C00542 V=800.0 PL=0
MOVL C00543 V=800.0 PL=0
MOVL C00544 V=800.0 PL=0
MOVL C00545 V=800.0 PL=0
MOVL C00546 V=800.0 PL=0
MOVL C00547 V=800.0 PL=0
MOVL C00548 V=800.0 PL=0
MOVL C00549 V=800.0 PL=0
MOVL C00550 V=800.0 PL=0
MOVL C00551 V=800.0 PL=0
MOVL C00552 V=800.0 PL=0
MOVL C00553 V=800.0 PL=0
MOVL C00554 V=800.0 PL=0
MOVL C00555 V=800.0 PL=0
MOVL C00556 V=800.0 PL=0
MOVL C00557 V=800.0 PL=0
MOVL C00558 V=800.0 PL=0
MOVL C00559 V=800.0 PL=0
MOVL C00560 V=800.0 PL=0
MOVL C00561 V=800.0 PL=0
MOVL C00562 V=800.0 PL=0
MOVL C00563 V=800.0 PL=0
MOVL C00564 V=800.0 PL=0
MOVL C00565 V=800.0 PL=0
MOVL C00566 V=800.0 PL=0
MOVL C00567 V=800.0 PL=0
MOVL C00568 V=800.0 PL=0
MOVL C00569 V=800.0 PL=0
MOVL C00570 V=800.0 PL=0
MOVL C00571 V=800.0 PL=0
MOVL C00572 V=800.0 PL=0
MOVL C00573 V=800.0 PL=0
MOVL C00574 V=800.0 PL=0
MOVL C00575 V=800.0 PL=0
MOVL C00576 V=800.0 PL=0
MOVL C00577 V=800.0 PL=0
MOVL C00578 V=800.0 PL=0
MOVL C00579 V=800.0 PL=0
MOVL C00580 V=800.0 PL=0
MOVL C00581 V=800.0 PL=0
MOVL C00582 V=800.0 PL=0
MOVL C00583 V=800.0 PL=0
MOVL C00584 V=800.0 PL=0
MOVL C00585 V=800.0 PL=0
MOVL C00586 V=800.0 PL=0
MOVL C00587 V=800.0 PL=0
MOVL C00588 V=800.0 PL=0
MOVL C00589 V=800.0 PL=0
MOVL C00590 V=800.0 PL=0
MOVL C00591 V=800.0 PL=0
MOVL C00592 V=800.0 PL=0
MOVL C00593 V=800.0 PL=0
MOVL C00594 V=800.0 PL=0
MOVL C00595 V=800.0 PL=0
MOVL C00596 V=800.0 PL=0
MOVL C00597 V=800.0 PL=0
MOVL C00598 V=800.0 PL=0
MOVL C00599 V=800.0 PL=0
MOVL C00600 V=800.0 PL=0
MOVL C00601 V=800.0 PL=0
MOVL C00602 V=800.0 PL=0
MOVL C00603 V=800.0 PL=0
MOVL C00604 V=800.0 PL=0
MOVL C00605 V=800.0 PL=0
MOVL C00606 V=800.0 PL=0
MOVL C00607 V=800.0 PL=0
MOVL C00608 V=800.0 PL=0
MOVL C00609 V=800.0 PL=0
MOVL C00610 V=800.0 PL=0
MOVL C00611 V=800.0 PL=0
MOVL C00612 V=800.0 PL=0
MOVL C00613 V=800.0 PL=0
MOVL C00614 V=800.0 PL=0
MOVL C00615 V=800.0 PL=0
MOVL C00616 V=800.0 PL=0
MOVL C00617 V=800.0 PL=0
MOVL C00618 V=800.0 PL=0
MOVL C00619 V=800.0 PL=0
MOVL C00620 V=800.0 PL=0
MOVL C00621 V=800.0 PL=0
MOVL C00622 V=800.0 PL=0
MOVL C00623 V=800.0 PL=0
MOVL C00624 V=800.0 PL=0
MOVL C00625 V=800.0 PL=0
MOVL C00626 V=800.0 PL=0
MOVL C00627 V=800.0 PL=0
MOVL C00628 V=800.0 PL=0
MOVL C00629 V=800.0 PL=0
MOVL C00630 V=800.0 PL=0
MOVL C00631 V=800.0 PL=0
MOVL C00632 V=800.0 PL=0
MOVL C00633 V=800.0 PL=0
MOVL C00634 V=800.0 PL=0
MOVL C00635 V=800.0 PL=0
MOVL C00636 V=800.0 PL=0
MOVL C00637 V=800.0 PL=0
MOVL C00638 V=800.0 PL=0
MOVL C00639 V=800.0 PL=0
MOVL C00640 V=800.0 PL=0
MOVL C00641 V=800.0 PL=0
MOVL C00642 V=800.0 PL=0
MOVL C00643 V=800.0 PL=0
MOVL C00644 V=800.0 PL=0
MOVL C00645 V=800.0 PL=0
MOVL C00646 V=800.0 PL=0
MOVL C00647 V=800.0 PL=0
MOVL C00648 V=800.0 PL=0
MOVL C00649 V=800.0 PL=0
MOVL C00650 V=800.0 PL=0
MOVL C00651 V=800.0 PL=0
MOVL C00652 V=800.0 PL=0
MOVL C00653 V=800.0 PL=0
MOVL C00654 V=800.0 PL=0
MOVL C00655 V=800.0 PL=0
MOVL C00656 V=800.0 PL=0
MOVL C00657 V=800.0 PL=0
MOVL C00658 V=800.0 PL=0
MOVL C00659 V=800.0 PL=0
MOVL C00660 V=800.0 PL=0
MOVL C00661 V=800.0 PL=0
MOVL C00662 V=800.0 PL=0
MOVL C00663 V=800.0 PL=0
MOVL C00664 V=800.0 PL=0
MOVL C00665 V=800.0 PL=0
MOVL C00666 V=800.0 PL=0
MOVL C00667 V=800.0 PL=0
MOVL C00668 V=800.0 PL=0
MOVL C00669 V=800.0 PL=0
MOVL C00670 V=800.0 PL=0
MOVL C00671 V=800.0 PL=0
MOVL C00672 V=800.0 PL=0
MOVL C00673 V=800.0 PL=0
MOVL C00674 V=800.0 PL=0
MOVL C00675 V=800.0 PL=0
MOVL C00676 V=800.0 PL=0
MOVL C00677 V=800.0 PL=0
MOVL C00678 V=800.0 PL=0
MOVL C00679 V=800.0 PL=0
MOVL C00680 V=800.0 PL=0
MOVL C00681 V=800.0 PL=0
MOVL C00682 V=800.0 PL=0
MOVL C00683 V=800.0 PL=0
MOVL C00684 V=800.0 PL=0
MOVL C00685 V=800.0 PL=0
MOVL C00686 V=800.0 PL=0
MOVL C00687 V=800.0 PL=0
MOVL C00688 V=800.0 PL=0
MOVL C00689 V=800.0 PL=0
MOVL C00690 V=800.0 PL=0
MOVL C00691 V=800.0 PL=0
MOVL C00692 V=800.0 PL=0
MOVL C00693 V=800.0 PL=0
MOVL C00694 V=800.0 PL=0
MOVL C00695 V=800.0 PL=0
MOVL C00696 V=800.0 PL=0
MOVL C00697 V=800.0 PL=0
MOVL C00698 V=800.0 PL=0
MOVL C00699 V=800.0 PL=0
MOVL C00700 V=800.0 PL=0
MOVL C00701 V=800.0 PL=0
MOVL C00702 V=800.0 PL=0
MOVL C00703 V=800.0 PL=0
MOVL C00704 V=800.0 PL=0
MOVL C00705 V=800.0 PL=0
MOVL C00706 V=800.0 PL=0
MOVL C00707 V=800.0 PL=0
MOVL C00708 V=800.0 PL=0
MOVL C00709 V=800.0 PL=0
MOVL C00710 V=800.0 PL=0
MOVL C00711 V=800.0 PL=0
MOVL C00712 V=800.0 PL=0
MOVL C00713 V=800.0 PL=0
MOVL C00714 V=800.0 PL=0
MOVL C00715 V=800.0 PL=0
MOVL C00716 V=800.0 PL=0
MOVL C00717 V=800.0 PL=0
MOVL C00718 V=800.0 PL=0
MOVL C00719 V=800.0 PL=0
MOVL C00720 V=800.0 PL=0
MOVL C00721 V=800.0 PL=0
MOVL C00722 V=800.0 PL=0
MOVL C00723 V=800.0 PL=0
MOVL C00724 V=800.0 PL=0
MOVL C00725 V=800.0 PL=0
MOVL C00726 V=800.0 PL=0
MOVL C00727 V=800.0 PL=0
MOVL C00728 V=800.0 PL=0
MOVL C00729 V=800.0 PL=0
MOVL C00730 V=800.0 PL=0
MOVL C00731 V=800.0 PL=0
MOVL C00732 V=800.0 PL=0
MOVL C00733 V=800.0 PL=0
MOVL C00734 V=800.0 PL=0
MOVL C00735 V=800.0 PL=0
MOVL C00736 V=800.0 PL=0
MOVL C00737 V=800.0 PL=0
MOVL C00738 V=800.0 PL=0
MOVL C00739 V=800.0 PL=0
MOVL C00740 V=800.0 PL=0
MOVL C00741 V=800.0 PL=0
MOVL C00742 V=800.0 PL=0
MOVL C00743 V=800.0 PL=0
MOVL C00744 V=800.0 PL=0
MOVL C00745 V=800.0 PL=0
MOVL C00746 V=800.0 PL=0
MOVL C00747 V=800.0 PL=0
MOVL C00748 V=800.0 PL=0
MOVL C00749 V=800.0 PL=0
MOVL C00750 V=800.0 PL=0
MOVL C00751 V=800.0 PL=0
MOVL C00752 V=800.0 PL=0
MOVL C00753 V=800.0 PL=0
MOVL C00754 V=800.0 PL=0
MOVL C00755 V=800.0 PL=0
MOVL C00756 V=800.0 PL=0
MOVL C00757 V=800.0 PL=0
MOVL C00758 V=800.0 PL=0
MOVL C00759 V=800.0 PL=0
MOVL C00760 V=800.0 PL=0
MOVL C00761 V=800.0 PL=0
MOVL C00762 V=800.0 PL=0
MOVL C00763 V=800.0 PL=0
MOVL C00764 V=800.0 PL=0
MOVL C00765 V=800.0 PL=0
MOVL C00766 V=800.0 PL=0
MOVL C00767 V=800.0 PL=0
MOVL C00768 V=800.0 PL=0
MOVL C00769 V=800.0 PL=0
MOVL C00770 V=800.0 PL=0
MOVL C00771 V=800.0 PL=0
MOVL C00772 V=800.0 PL=0
MOVL C00773 V=800.0 PL=0
MOVL C00774 V=800.0 PL=0
MOVL C00775 V=800.0 PL=0
MOVL C00776 V=800.0 PL=0
MOVL C00777 V=800.0 PL=0
MOVL C00778 V=800.0 PL=0
MOVL C00779 V=800.0 PL=0
MOVL C00780 V=800.0 PL=0
MOVL C00781 V=800.0 PL=0
MOVL C00782 V=800.0 PL=0
MOVL C00783 V=800.0 PL=0
MOVL C00784 V=800.0 PL=0
MOVL C00785 V=800.0 PL=0
MOVL C00786 V=800.0 PL=0
MOVL C00787 V=800.0 PL=0
MOVL C00788 V=800.0 PL=0
MOVL C00789 V=800.0 PL=0
MOVL C00790 V=800.0 PL=0
MOVL C00791 V=800.0 PL=0
MOVL C00792 V=800.0 PL=0
MOVL C00793 V=800.0 PL=0
MOVL C00794 V=800.0 PL=0
MOVL C00795 V=800.0 PL=0
MOVL C00796 V=800.0 PL=0
MOVL C00797 V=800.0 PL=0
MOVL C00798 V=800.0 PL=0
MOVL C00799 V=800.0 PL=0
MOVL C00800 V=800.0 PL=0
MOVL C00801 V=800.0 PL=0
MOVL C00802 V=800.0 PL=0
MOVL C00803 V=800.0 PL=0
MOVL C00804 V=800.0 PL=0
MOVL C00805 V=800.0 PL=0
MOVL C00806 V=800.0 PL=0
MOVL C00807 V=800.0 PL=0
MOVL C00808 V=800.0 PL=0
MOVL C00809 V=800.0 PL=0
MOVL C00810 V=800.0 PL=0
MOVL C00811 V=800.0 PL=0
MOVL C00812 V=800.0 PL=0
MOVL C00813 V=800.0 PL=0
MOVL C00814 V=800.0 PL=0
MOVL C00815 V=800.0 PL=0
MOVL C00816 V=800.0 PL=0
MOVL C00817 V=800.0 PL=0
MOVL C00818 V=800.0 PL=0
MOVL C00819 V=800.0 PL=0
MOVL C00820 V=800.0 PL=0
MOVL C00821 V=800.0 PL=0
MOVL C00822 V=800.0 PL=0
MOVL C00823 V=800.0 PL=0
MOVL C00824 V=800.0 PL=0
MOVL C00825 V=800.0 PL=0
MOVL C00826 V=800.0 PL=0
MOVL C00827 V=800.0 PL=0
MOVL C00828 V=800.0 PL=0
MOVL C00829 V=800.0 PL=0
MOVL C00830 V=800.0 PL=0
MOVL C00831 V=800.0 PL=0
MOVL C00832 V=800.0 PL=0
MOVL C00833 V=800.0 PL=0
MOVL C00834 V=800.0 PL=0
MOVL C00835 V=800.0 PL=0
MOVL C00836 V=800.0 PL=0
MOVL C00837 V=800.0 PL=0
MOVL C00838 V=800.0 PL=0
MOVL C00839 V=800.0 PL=0
MOVL C00840 V=800.0 PL=0
MOVL C00841 V=800.0 PL=0
MOVL C00842 V=800.0 PL=0
MOVL C00843 V=800.0 PL=0
MOVL C00844 V=800.0 PL=0
MOVL C00845 V=800.0 PL=0
MOVL C00846 V=800.0 PL=0
MOVL C00847 V=800.0 PL=0
MOVL C00848 V=800.0 PL=0
MOVL C00849 V=800.0 PL=0
MOVL C00850 V=800.0 PL=0
MOVL C00851 V=800.0 PL=0
MOVL C00852 V=800.0 PL=0
MOVL C00853 V=800.0 PL=0
MOVL C00854 V=800.0 PL=0
MOVL C00855 V=800.0 PL=0
MOVL C00856 V=800.0 PL=0
MOVL C00857 V=800.0 PL=0
MOVL C00858 V=800.0 PL=0
MOVL C00859 V=800.0 PL=0
MOVL C00860 V=800.0 PL=0
MOVL C00861 V=800.0 PL=0
MOVL C00862 V=800.0 PL=0
MOVL C00863 V=800.0 PL=0
MOVL C00864 V=800.0 PL=0
MOVL C00865 V=800.0 PL=0
MOVL C00866 V=800.0 PL=0
MOVL C00867 V=800.0 PL=0
MOVL C00868 V=800.0 PL=0
MOVL C00869 V=800.0 PL=0
MOVL C00870 V=800.0 PL=0
MOVL C00871 V=800.0 PL=0
MOVL C00872 V=800.0 PL=0
MOVL C00873 V=800.0 PL=0
MOVL C00874 V=800.0 PL=0
MOVL C00875 V=800.0 PL=0
MOVL C00876 V=800.0 PL=0
MOVL C00877 V=800.0 PL=0
MOVL C00878 V=800.0 PL=0
MOVL C00879 V=800.0 PL=0
MOVL C00880 V=800.0 PL=0
MOVL C00881 V=800.0 PL=0
MOVL C00882 V=800.0 PL=0
MOVL C00883 V=800.0 PL=0
MOVL C00884 V=800.0 PL=0
MOVL C00885 V=800.0 PL=0
MOVL C00886 V=800.0 PL=0
MOVL C00887 V=800.0 PL=0
MOVL C00888 V=800.0 PL=0
MOVL C00889 V=800.0 PL=0
MOVL C00890 V=800.0 PL=0
MOVL C00891 V=800.0 PL=0
MOVL C00892 V=800.0 PL=0
MOVL C00893 V=800.0 PL=0
MOVL C00894 V=800.0 PL=0
MOVL C00895 V=800.0 PL=0
MOVL C00896 V=800.0 PL=0
MOVL C00897 V=800.0 PL=0
MOVL C00898 V=800.0 PL=0
MOVL C00899 V=800.0 PL=0
MOVL C00900 V=800.0 PL=0
MOVL C00901 V=800.0 PL=0
MOVL C00902 V=800.0 PL=0
MOVL C00903 V=800.0 PL=0
MOVL C00904 V=800.0 PL=0
MOVL C00905 V=800.0 PL=0
MOVL C00906 V=800.0 PL=0
MOVL C00907 V=800.0 PL=0
MOVL C00908 V=800.0 PL=0
MOVL C00909 V=800.0 PL=0
MOVL C00910 V=800.0 PL=0
MOVL C00911 V=800.0 PL=0
MOVL C00912 V=800.0 PL=0
MOVL C00913 V=800.0 PL=0
MOVL C00914 V=800.0 PL=0
MOVL C00915 V=800.0 PL=0
MOVL C00916 V=800.0 PL=0
MOVL C00917 V=800.0 PL=0
MOVL C00918 V=800.0 PL=0
MOVL C00919 V=800.0 PL=0
MOVL C00920 V=800.0 PL=0
MOVL C00921 V=800.0 PL=0
MOVL C00922 V=800.0 PL=0
MOVL C00923 V=800.0 PL=0
MOVL C00924 V=800.0 PL=0
MOVL C00925 V=800.0 PL=0
MOVL C00926 V=800.0 PL=0
MOVL C00927 V=800.0 PL=0
MOVL C00928 V=800.0 PL=0
MOVL C00929 V=800.0 PL=0
MOVL C00930 V=800.0 PL=0
MOVL C00931 V=800.0 PL=0
MOVL C00932 V=800.0 PL=0
MOVL C00933 V=800.0 PL=0
MOVL C00934 V=800.0 PL=0
MOVL C00935 V=800.0 PL=0
MOVL C00936 V=800.0 PL=0
MOVL C00937 V=800.0 PL=0
MOVL C00938 V=800.0 PL=0
MOVL C00939 V=800.0 PL=0
MOVL C00940 V=800.0 PL=0
MOVL C00941 V=800.0 PL=0
MOVL C00942 V=800.0 PL=0
MOVL C00943 V=800.0 PL=0
MOVL C00944 V=800.0 PL=0
MOVL C00945 V=800.0 PL=0
MOVL C00946 V=800.0 PL=0
MOVL C00947 V=800.0 PL=0
MOVL C00948 V=800.0 PL=0
MOVL C00949 V=800.0 PL=0
MOVL C00950 V=800.0 PL=0
MOVL C00951 V=800.0 PL=0
MOVL C00952 V=800.0 PL=0
MOVL C00953 V=800.0 PL=0
MOVL C00954 V=800.0 PL=0
MOVL C00955 V=800.0 PL=0
MOVL C00956 V=800.0 PL=0
MOVL C00957 V=800.0 PL=0
MOVL C00958 V=800.0 PL=0
MOVL C00959 V=800.0 PL=0
MOVL C00960 V=800.0 PL=0
MOVL C00961 V=800.0 PL=0
MOVL C00962 V=800.0 PL=0
MOVL C00963 V=800.0 PL=0
MOVL C00964 V=800.0 PL=0
MOVL C00965 V=800.0 PL=0
MOVL C00966 V=800.0 PL=0
MOVL C00967 V=800.0 PL=0
MOVL C00968 V=800.0 PL=0
MOVL C00969 V=800.0 PL=0
MOVL C00970 V=800.0 PL=0
MOVL C00971 V=800.0 PL=0
MOVL C00972 V=800.0 PL=0
MOVL C00973 V=800.0 PL=0
MOVL C00974 V=800.0 PL=0
MOVL C00975 V=800.0 PL=0
MOVL C00976 V=800.0 PL=0
MOVL C00977 V=800.0 PL=0
MOVL C00978 V=800.0 PL=0
MOVL C00979 V=800.0 PL=0
MOVL C00980 V=800.0 PL=0
MOVL C00981 V=800.0 PL=0
MOVL C00982 V=800.0 PL=0
MOVL C00983 V=800.0 PL=0
MOVL C00984 V=800.0 PL=0
MOVL C00985 V=800.0 PL=0
MOVL C00986 V=800.0 PL=0
MOVL C00987 V=800.0 PL=0
MOVL C00988 V=800.0 PL=0
MOVL C00989 V=800.0 PL=0
MOVL C00990 V=800.0 PL=0
MOVL C00991 V=800.0 PL=0
MOVL C00992 V=800.0 PL=0
MOVL C00993 V=800.0 PL=0
MOVL C00994 V=800.0 PL=0
MOVL C00995 V=800.0 PL=0
MOVL C00996 V=800.0 PL=0
MOVL C00997 V=800.0 PL=0
MOVL C00998 V=800.0 PL=0
MOVL C00999 V=800.0 PL=0
MOVL C01000 V=800.0 PL=0
MOVL C01001 V=800.0 PL=0
MOVL C01002 V=800.0 PL=0
MOVL C01003 V=800.0 PL=0
MOVL C01004 V=800.0 PL=0
MOVL C01005 V=800.0 PL=0
MOVL C01006 V=800.0 PL=0
MOVL C01007 V=800.0 PL=0
MOVL C01008 V=800.0 PL=0
MOVL C01009 V=800.0 PL=0
MOVL C01010 V=800.0 PL=0
MOVL C01011 V=800.0 PL=0
MOVL C01012 V=800.0 PL=0
MOVL C01013 V=800.0 PL=0
MOVL C01014 V=800.0 PL=0
MOVL C01015 V=800.0 PL=0
MOVL C01016 V=800.0 PL=0
MOVL C01017 V=800.0 PL=0
MOVL C01018 V=800.0 PL=0
MOVL C01019 V=800.0 PL=0
MOVL C01020 V=800.0 PL=0
MOVL C01021 V=800.0 PL=0
MOVL C01022 V=800.0 PL=0
MOVL C01023 V=800.0 PL=0
MOVL C01024 V=800.0 PL=0
MOVL C01025 V=800.0 PL=0
MOVL C01026 V=800.0 PL=0
MOVL C01027 V=800.0 PL=0
MOVL C01028 V=800.0 PL=0
MOVL C01029 V=800.0 PL=0
MOVL C01030 V=800.0 PL=0
MOVL C01031 V=800.0 PL=0
MOVL C01032 V=800.0 PL=0
MOVL C01033 V=800.0 PL=0
MOVL C01034 V=800.0 PL=0
MOVL C01035 V=800.0 PL=0
MOVL C01036 V=800.0 PL=0
MOVL C01037 V=800.0 PL=0
MOVL C01038 V=800.0 PL=0
MOVL C01039 V=800.0 PL=0
MOVL C01040 V=800.0 PL=0
MOVL C01041 V=800.0 PL=0
MOVL C01042 V=800.0 PL=0
MOVL C01043 V=800.0 PL=0
MOVL C01044 V=800.0 PL=0
MOVL C01045 V=800.0 PL=0
MOVL C01046 V=800.0 PL=0
MOVL C01047 V=800.0 PL=0
MOVL C01048 V=800.0 PL=0
MOVL C01049 V=800.0 PL=0
MOVL C01050 V=800.0 PL=0
MOVL C01051 V=800.0 PL=0
MOVL C01052 V=800.0 PL=0
MOVL C01053 V=800.0 PL=0
MOVL C01054 V=800.0 PL=0
MOVL C01055 V=800.0 PL=0
MOVL C01056 V=800.0 PL=0
MOVL C01057 V=800.0 PL=0
MOVL C01058 V=800.0 PL=0
MOVL C01059 V=800.0 PL=0
MOVL C01060 V=800.0 PL=0
MOVL C01061 V=800.0 PL=0
MOVL C01062 V=800.0 PL=0
MOVL C01063 V=800.0 PL=0
MOVL C01064 V=800.0 PL=0
MOVL C01065 V=800.0 PL=0
MOVL C01066 V=800.0 PL=0
MOVL C01067 V=800.0 PL=0
MOVL C01068 V=800.0 PL=0
MOVL C01069 V=800.0 PL=0
MOVL C01070 V=800.0 PL=0
MOVL C01071 V=800.0 PL=0
MOVL C01072 V=800.0 PL=0
MOVL C01073 V=800.0 PL=0
MOVL C01074 V=800.0 PL=0
MOVL C01075 V=800.0 PL=0
MOVL C01076 V=800.0 PL=0
MOVL C01077 V=800.0 PL=0
MOVL C01078 V=800.0 PL=0
MOVL C01079 V=800.0 PL=0
MOVL C01080 V=800.0 PL=0
MOVL C01081 V=800.0 PL=0
MOVL C01082 V=800.0 PL=0
MOVL C01083 V=800.0 PL=0
MOVL C01084 V=800.0 PL=0
MOVL C01085 V=800.0 PL=0
MOVL C01086 V=800.0 PL=0
MOVL C01087 V=800.0 PL=0
MOVL C01088 V=800.0 PL=0
MOVL C01089 V=800.0 PL=0
MOVL C01090 V=800.0 PL=0
MOVL C01091 V=800.0 PL=0
MOVL C01092 V=800.0 PL=0
MOVL C01093 V=800.0 PL=0
MOVL C01094 V=800.0 PL=0
MOVL C01095 V=800.0 PL=0
MOVL C01096 V=800.0 PL=0
MOVL C01097 V=800.0 PL=0
MOVL C01098 V=800.0 PL=0
MOVL C01099 V=800.0 PL=0
MOVL C01100 V=800.0 PL=0
MOVL C01101 V=800.0 PL=0
MOVL C01102 V=800.0 PL=0
MOVL C01103 V=800.0 PL=0
MOVL C01104 V=800.0 PL=0
MOVL C01105 V=800.0 PL=0
MOVL C01106 V=800.0 PL=0
MOVL C01107 V=800.0 PL=0
MOVL C01108 V=800.0 PL=0
MOVL C01109 V=800.0 PL=0
MOVL C01110 V=800.0 PL=0
MOVL C01111 V=800.0 PL=0
MOVL C01112 V=800.0 PL=0
MOVL C01113 V=800.0 PL=0
MOVL C01114 V=800.0 PL=0
MOVL C01115 V=800.0 PL=0
MOVL C01116 V=800.0 PL=0
MOVL C01117 V=800.0 PL=0
MOVL C01118 V=800.0 PL=0
MOVL C01119 V=800.0 PL=0
MOVL C01120 V=800.0 PL=0
MOVL C01121 V=800.0 PL=0
MOVL C01122 V=800.0 PL=0
MOVL C01123 V=800.0 PL=0
MOVL C01124 V=800.0 PL=0
MOVL C01125 V=800.0 PL=0
MOVL C01126 V=800.0 PL=0
MOVL C01127 V=800.0 PL=0
MOVL C01128 V=800.0 PL=0
MOVL C01129 V=800.0 PL=0
MOVL C01130 V=800.0 PL=0
MOVL C01131 V=800.0 PL=0
MOVL C01132 V=800.0 PL=0
MOVL C01133 V=800.0 PL=0
MOVL C01134 V=800.0 PL=0
MOVL C01135 V=800.0 PL=0
MOVL C01136 V=800.0 PL=0
MOVL C01137 V=800.0 PL=0
MOVL C01138 V=800.0 PL=0
MOVL C01139 V=800.0 PL=0
MOVL C01140 V=800.0 PL=0
MOVL C01141 V=800.0 PL=0
MOVL C01142 V=800.0 PL=0
MOVL C01143 V=800.0 PL=0
MOVL C01144 V=800.0 PL=0
MOVL C01145 V=800.0 PL=0
MOVL C01146 V=800.0 PL=0
MOVL C01147 V=800.0 PL=0
MOVL C01148 V=800.0 PL=0
MOVL C01149 V=800.0 PL=0
MOVL C01150 V=800.0 PL=0
MOVL C01151 V=800.0 PL=0
MOVL C01152 V=800.0 PL=0
MOVL C01153 V=800.0 PL=0
MOVL C01154 V=800.0 PL=0
MOVL C01155 V=800.0 PL=0
MOVL C01156 V=800.0 PL=0
MOVL C01157 V=800.0 PL=0
MOVL C01158 V=800.0 PL=0
MOVL C01159 V=800.0 PL=0
MOVL C01160 V=800.0 PL=0
MOVL C01161 V=800.0 PL=0
MOVL C01162 V=800.0 PL=0
MOVL C01163 V=800.0 PL=0
MOVL C01164 V=800.0 PL=0
MOVL C01165 V=800.0 PL=0
MOVL C01166 V=800.0 PL=0
MOVL C01167 V=800.0 PL=0
MOVL C01168 V=800.0 PL=0
MOVL C01169 V=800.0 PL=0
MOVL C01170 V=800.0 PL=0
MOVL C01171 V=800.0 PL=0
MOVL C01172 V=800.0 PL=0
MOVL C01173 V=800.0 PL=0
MOVL C01174 V=800.0 PL=0
MOVL C01175 V=800.0 PL=0
MOVL C01176 V=800.0 PL=0
MOVL C01177 V=800.0 PL=0
MOVL C01178 V=800.0 PL=0
MOVL C01179 V=800.0 PL=0
MOVL C01180 V=800.0 PL=0
MOVL C01181 V=800.0 PL=0
MOVL C01182 V=800.0 PL=0
MOVL C01183 V=800.0 PL=0
MOVL C01184 V=800.0 PL=0
MOVL C01185 V=800.0 PL=0
MOVL C01186 V=800.0 PL=0
MOVL C01187 V=800.0 PL=0
MOVL C01188 V=800.0 PL=0
MOVL C01189 V=800.0 PL=0
MOVL C01190 V=800.0 PL=0
MOVL C01191 V=800.0 PL=0
MOVL C01192 V=800.0 PL=0
MOVL C01193 V=800.0 PL=0
MOVL C01194 V=800.0 PL=0
MOVL C01195 V=800.0 PL=0
MOVL C01196 V=800.0 PL=0
MOVL C01197 V=800.0 PL=0
MOVL C01198 V=800.0 PL=0
MOVL C01199 V=800.0 PL=0
MOVL C01200 V=800.0 PL=0
MOVL C01201 V=800.0 PL=0
MOVL C01202 V=800.0 PL=0
MOVL C01203 V=800.0 PL=0
MOVL C01204 V=800.0 PL=0
MOVL C01205 V=800.0 PL=0
MOVL C01206 V=800.0 PL=0
MOVL C01207 V=800.0 PL=0
MOVL C01208 V=800.0 PL=0
MOVL C01209 V=800.0 PL=0
MOVL C01210 V=800.0 PL=0
MOVL C01211 V=800.0 PL=0
MOVL C01212 V=800.0 PL=0
MOVL C01213 V=800.0 PL=0
MOVL C01214 V=800.0 PL=0
MOVL C01215 V=800.0 PL=0
MOVL C01216 V=800.0 PL=0
MOVL C01217 V=800.0 PL=0
MOVL C01218 V=800.0 PL=0
MOVL C01219 V=800.0 PL=0
MOVL C01220 V=800.0 PL=0
MOVL C01221 V=800.0 PL=0
MOVL C01222 V=800.0 PL=0
MOVL C01223 V=800.0 PL=0
MOVL C01224 V=800.0 PL=0
MOVL C01225 V=800.0 PL=0
MOVL C01226 V=800.0 PL=0
MOVL C01227 V=800.0 PL=0
MOVL C01228 V=800.0 PL=0
MOVL C01229 V=800.0 PL=0
MOVL C01230 V=800.0 PL=0
MOVL C01231 V=800.0 PL=0
MOVL C01232 V=800.0 PL=0
MOVL C01233 V=800.0 PL=0
MOVL C01234 V=800.0 PL=0
MOVL C01235 V=800.0 PL=0
MOVL C01236 V=800.0 PL=0
MOVL C01237 V=800.0 PL=0
MOVL C01238 V=800.0 PL=0
MOVL C01239 V=800.0 PL=0
MOVL C01240 V=800.0 PL=0
MOVL C01241 V=800.0 PL=0
MOVL C01242 V=800.0 PL=0
MOVL C01243 V=800.0 PL=0
MOVL C01244 V=800.0 PL=0
MOVL C01245 V=800.0 PL=0
MOVL C01246 V=800.0 PL=0
MOVL C01247 V=800.0 PL=0
MOVL C01248 V=800.0 PL=0
MOVL C01249 V=800.0 PL=0
MOVL C01250 V=800.0 PL=0
MOVL C01251 V=800.0 PL=0
MOVL C01252 V=800.0 PL=0
MOVL C01253 V=800.0 PL=0
MOVL C01254 V=800.0 PL=0
MOVL C01255 V=800.0 PL=0
MOVL C01256 V=800.0 PL=0
MOVL C01257 V=800.0 PL=0
MOVL C01258 V=800.0 PL=0
MOVL C01259 V=800.0 PL=0
MOVL C01260 V=800.0 PL=0
MOVL C01261 V=800.0 PL=0
MOVL C01262 V=800.0 PL=0
MOVL C01263 V=800.0 PL=0
MOVL C01264 V=800.0 PL=0
MOVL C01265 V=800.0 PL=0
MOVL C01266 V=800.0 PL=0
MOVL C01267 V=800.0 PL=0
MOVL C01268 V=800.0 PL=0
MOVL C01269 V=800.0 PL=0
MOVL C01270 V=800.0 PL=0
MOVL C01271 V=800.0 PL=0
MOVL C01272 V=800.0 PL=0
MOVL C01273 V=800.0 PL=0
MOVL C01274 V=800.0 PL=0
MOVL C01275 V=800.0 PL=0
MOVL C01276 V=800.0 PL=0
MOVL C01277 V=800.0 PL=0
MOVL C01278 V=800.0 PL=0
MOVL C01279 V=800.0 PL=0
MOVL C01280 V=800.0 PL=0
MOVL C01281 V=800.0 PL=0
MOVL C01282 V=800.0 PL=0
MOVL C01283 V=800.0 PL=0
MOVL C01284 V=800.0 PL=0
MOVL C01285 V=800.0 PL=0
MOVL C01286 V=800.0 PL=0
MOVL C01287 V=800.0 PL=0
MOVL C01288 V=800.0 PL=0
MOVL C01289 V=800.0 PL=0
MOVL C01290 V=800.0 PL=0
MOVL C01291 V=800.0 PL=0
MOVL C01292 V=800.0 PL=0
MOVL C01293 V=800.0 PL=0
MOVL C01294 V=800.0 PL=0
MOVL C01295 V=800.0 PL=0
MOVL C01296 V=800.0 PL=0
MOVL C01297 V=800.0 PL=0
MOVL C01298 V=800.0 PL=0
MOVL C01299 V=800.0 PL=0
MOVL C01300 V=800.0 PL=0
MOVL C01301 V=800.0 PL=0
MOVL C01302 V=800.0 PL=0
MOVL C01303 V=800.0 PL=0
MOVL C01304 V=800.0 PL=0
MOVL C01305 V=800.0 PL=0
MOVL C01306 V=800.0 PL=0
MOVL C01307 V=800.0 PL=0
MOVL C01308 V=800.0 PL=0
MOVL C01309 V=800.0 PL=0
MOVL C01310 V=800.0 PL=0
MOVL C01311 V=800.0 PL=0
MOVL C01312 V=800.0 PL=0
MOVL C01313 V=800.0 PL=0
MOVL C01314 V=800.0 PL=0
MOVL C01315 V=800.0 PL=0
MOVL C01316 V=800.0 PL=0
MOVL C01317 V=800.0 PL=0
MOVL C01318 V=800.0 PL=0
MOVL C01319 V=800.0 PL=0
MOVL C01320 V=800.0 PL=0
MOVL C01321 V=800.0 PL=0
MOVL C01322 V=800.0 PL=0
MOVL C01323 V=800.0 PL=0
MOVL C01324 V=800.0 PL=0
MOVL C01325 V=800.0 PL=0
MOVL C01326 V=800.0 PL=0
MOVL C01327 V=800.0 PL=0
MOVL C01328 V=800.0 PL=0
MOVL C01329 V=800.0 PL=0
MOVL C01330 V=800.0 PL=0
MOVL C01331 V=800.0 PL=0
MOVL C01332 V=800.0 PL=0
MOVL C01333 V=800.0 PL=0
MOVL C01334 V=800.0 PL=0
MOVL C01335 V=800.0 PL=0
MOVL C01336 V=800.0 PL=0
MOVL C01337 V=800.0 PL=0
MOVL C01338 V=800.0 PL=0
MOVL C01339 V=800.0 PL=0
MOVL C01340 V=800.0 PL=0
MOVL C01341 V=800.0 PL=0
MOVL C01342 V=800.0 PL=0
MOVL C01343 V=800.0 PL=0
MOVL C01344 V=800.0 PL=0
MOVL C01345 V=800.0 PL=0
MOVL C01346 V=800.0 PL=0
MOVL C01347 V=800.0 PL=0
MOVL C01348 V=800.0 PL=0
MOVL C01349 V=800.0 PL=0
MOVL C01350 V=800.0 PL=0
MOVL C01351 V=800.0 PL=0
MOVL C01352 V=800.0 PL=0
MOVL C01353 V=800.0 PL=0
MOVL C01354 V=800.0 PL=0
MOVL C01355 V=800.0 PL=0
MOVL C01356 V=800.0 PL=0
MOVL C01357 V=800.0 PL=0
MOVL C01358 V=800.0 PL=0
MOVL C01359 V=800.0 PL=0
MOVL C01360 V=800.0 PL=0
MOVL C01361 V=800.0 PL=0
MOVL C01362 V=800.0 PL=0
MOVL C01363 V=800.0 PL=0
MOVL C01364 V=800.0 PL=0
MOVL C01365 V=800.0 PL=0
MOVL C01366 V=800.0 PL=0
MOVL C01367 V=800.0 PL=0
MOVL C01368 V=800.0 PL=0
MOVL C01369 V=800.0 PL=0
MOVL C01370 V=800.0 PL=0
MOVL C01371 V=800.0 PL=0
MOVL C01372 V=800.0 PL=0
MOVL C01373 V=800.0 PL=0
MOVL C01374 V=800.0 PL=0
MOVL C01375 V=800.0 PL=0
MOVL C01376 V=800.0 PL=0
MOVL C01377 V=800.0 PL=0
MOVL C01378 V=800.0 PL=0
MOVL C01379 V=800.0 PL=0
MOVL C01380 V=800.0 PL=0
MOVL C01381 V=800.0 PL=0
MOVL C01382 V=800.0 PL=0
MOVL C01383 V=800.0 PL=0
MOVL C01384 V=800.0 PL=0
MOVL C01385 V=800.0 PL=0
MOVL C01386 V=800.0 PL=0
MOVL C01387 V=800.0 PL=0
MOVL C01388 V=800.0 PL=0
MOVL C01389 V=800.0 PL=0
MOVL C01390 V=800.0 PL=0
MOVL C01391 V=800.0 PL=0
MOVL C01392 V=800.0 PL=0
MOVL C01393 V=800.0 PL=0
MOVL C01394 V=800.0 PL=0
MOVL C01395 V=800.0 PL=0
MOVL C01396 V=800.0 PL=0
MOVL C01397 V=800.0 PL=0
MOVL C01398 V=800.0 PL=0
MOVL C01399 V=800.0 PL=0
MOVL C01400 V=800.0 PL=0
MOVL C01401 V=800.0 PL=0
MOVL C01402 V=800.0 PL=0
MOVL C01403 V=800.0 PL=0
MOVL C01404 V=800.0 PL=0
MOVL C01405 V=800.0 PL=0
MOVL C01406 V=800.0 PL=0
MOVL C01407 V=800.0 PL=0
MOVL C01408 V=800.0 PL=0
MOVL C01409 V=800.0 PL=0
MOVL C01410 V=800.0 PL=0
MOVL C01411 V=800.0 PL=0
MOVL C01412 V=800.0 PL=0
MOVL C01413 V=800.0 PL=0
MOVL C01414 V=800.0 PL=0
MOVL C01415 V=800.0 PL=0
MOVL C01416 V=800.0 PL=0
MOVL C01417 V=800.0 PL=0
MOVL C01418 V=800.0 PL=0
MOVL C01419 V=800.0 PL=0
MOVL C01420 V=800.0 PL=0
MOVL C01421 V=800.0 PL=0
MOVL C01422 V=800.0 PL=0
MOVL C01423 V=800.0 PL=0
MOVL C01424 V=800.0 PL=0
MOVL C01425 V=800.0 PL=0
MOVL C01426 V=800.0 PL=0
MOVL C01427 V=800.0 PL=0
MOVL C01428 V=800.0 PL=0
MOVL C01429 V=800.0 PL=0
MOVL C01430 V=800.0 PL=0
MOVL C01431 V=800.0 PL=0
MOVL C01432 V=800.0 PL=0
MOVL C01433 V=800.0 PL=0
MOVL C01434 V=800.0 PL=0
MOVL C01435 V=800.0 PL=0
MOVL C01436 V=800.0 PL=0
MOVL C01437 V=800.0 PL=0
MOVL C01438 V=800.0 PL=0
MOVL C01439 V=800.0 PL=0
MOVL C01440 V=800.0 PL=0
MOVL C01441 V=800.0 PL=0
MOVL C01442 V=800.0 PL=0
MOVL C01443 V=800.0 PL=0
MOVL C01444 V=800.0 PL=0
MOVL C01445 V=800.0 PL=0
MOVL C01446 V=800.0 PL=0
MOVL C01447 V=800.0 PL=0
MOVL C01448 V=800.0 PL=0
MOVL C01449 V=800.0 PL=0
MOVL C01450 V=800.0 PL=0
MOVL C01451 V=800.0 PL=0
MOVL C01452 V=800.0 PL=0
MOVL C01453 V=800.0 PL=0
MOVL C01454 V=800.0 PL=0
MOVL C01455 V=800.0 PL=0
MOVL C01456 V=800.0 PL=0
MOVL C01457 V=800.0 PL=0
MOVL C01458 V=800.0 PL=0
MOVL C01459 V=800.0 PL=0
MOVL C01460 V=800.0 PL=0
MOVL C01461 V=800.0 PL=0
MOVL C01462 V=800.0 PL=0
MOVL C01463 V=800.0 PL=0
MOVL C01464 V=800.0 PL=0
MOVL C01465 V=800.0 PL=0
MOVL C01466 V=800.0 PL=0
MOVL C01467 V=800.0 PL=0
MOVL C01468 V=800.0 PL=0
MOVL C01469 V=800.0 PL=0
MOVL C01470 V=800.0 PL=0
MOVL C01471 V=800.0 PL=0
MOVL C01472 V=800.0 PL=0
MOVL C01473 V=800.0 PL=0
MOVL C01474 V=800.0 PL=0
MOVL C01475 V=800.0 PL=0
MOVL C01476 V=800.0 PL=0
MOVL C01477 V=800.0 PL=0
MOVL C01478 V=800.0 PL=0
MOVL C01479 V=800.0 PL=0
MOVL C01480 V=800.0 PL=0
MOVL C01481 V=800.0 PL=0
MOVL C01482 V=800.0 PL=0
MOVL C01483 V=800.0 PL=0
MOVL C01484 V=800.0 PL=0
MOVL C01485 V=800.0 PL=0
MOVL C01486 V=800.0 PL=0
MOVL C01487 V=800.0 PL=0
MOVL C01488 V=800.0 PL=0
MOVL C01489 V=800.0 PL=0
MOVL C01490 V=800.0 PL=0
MOVL C01491 V=800.0 PL=0
MOVL C01492 V=800.0 PL=0
MOVL C01493 V=800.0 PL=0
MOVL C01494 V=800.0 PL=0
MOVL C01495 V=800.0 PL=0
MOVL C01496 V=800.0 PL=0
MOVL C01497 V=800.0 PL=0
MOVL C01498 V=800.0 PL=0
MOVL C01499 V=800.0 PL=0
MOVL C01500 V=800.0 PL=0
MOVL C01501 V=800.0 PL=0
MOVL C01502 V=800.0 PL=0
MOVL C01503 V=800.0 PL=0
MOVL C01504 V=800.0 PL=0
MOVL C01505 V=800.0 PL=0
MOVL C01506 V=800.0 PL=0
MOVL C01507 V=800.0 PL=0
MOVL C01508 V=800.0 PL=0
MOVL C01509 V=800.0 PL=0
MOVL C01510 V=800.0 PL=0
MOVL C01511 V=800.0 PL=0
MOVL C01512 V=800.0 PL=0
MOVL C01513 V=800.0 PL=0
MOVL C01514 V=800.0 PL=0
MOVL C01515 V=800.0 PL=0
MOVL C01516 V=800.0 PL=0
MOVL C01517 V=800.0 PL=0
MOVL C01518 V=800.0 PL=0
MOVL C01519 V=800.0 PL=0
MOVL C01520 V=800.0 PL=0
MOVL C01521 V=800.0 PL=0
MOVL C01522 V=800.0 PL=0
MOVL C01523 V=800.0 PL=0
MOVL C01524 V=800.0 PL=0
MOVL C01525 V=800.0 PL=0
MOVL C01526 V=800.0 PL=0
MOVL C01527 V=800.0 PL=0
MOVL C01528 V=800.0 PL=0
MOVL C01529 V=800.0 PL=0
MOVL C01530 V=800.0 PL=0
MOVL C01531 V=800.0 PL=0
MOVL C01532 V=800.0 PL=0
MOVL C01533 V=800.0 PL=0
MOVL C01534 V=800.0 PL=0
MOVL C01535 V=800.0 PL=0
MOVL C01536 V=800.0 PL=0
MOVL C01537 V=800.0 PL=0
MOVL C01538 V=800.0 PL=0
MOVL C01539 V=800.0 PL=0
MOVL C01540 V=800.0 PL=0
MOVL C01541 V=800.0 PL=0
MOVL C01542 V=800.0 PL=0
MOVL C01543 V=800.0 PL=0
MOVL C01544 V=800.0 PL=0
MOVL C01545 V=800.0 PL=0
MOVL C01546 V=800.0 PL=0
MOVL C01547 V=800.0 PL=0
MOVL C01548 V=800.0 PL=0
MOVL C01549 V=800.0 PL=0
MOVL C01550 V=800.0 PL=0
MOVL C01551 V=800.0 PL=0
MOVL C01552 V=800.0 PL=0
MOVL C01553 V=800.0 PL=0
MOVL C01554 V=800.0 PL=0
MOVL C01555 V=800.0 PL=0
MOVL C01556 V=800.0 PL=0
MOVL C01557 V=800.0 PL=0
MOVL C01558 V=800.0 PL=0
MOVL C01559 V=800.0 PL=0
MOVL C01560 V=800.0 PL=0
MOVL C01561 V=800.0 PL=0
MOVL C01562 V=800.0 PL=0
MOVL C01563 V=800.0 PL=0
MOVL C01564 V=800.0 PL=0
MOVL C01565 V=800.0 PL=0
MOVL C01566 V=800.0 PL=0
MOVL C01567 V=800.0 PL=0
MOVL C01568 V=800.0 PL=0
MOVL C01569 V=800.0 PL=0
MOVL C01570 V=800.0 PL=0
MOVL C01571 V=800.0 PL=0
MOVL C01572 V=800.0 PL=0
MOVL C01573 V=800.0 PL=0
MOVL C01574 V=800.0 PL=0
MOVL C01575 V=800.0 PL=0
MOVL C01576 V=800.0 PL=0
MOVL C01577 V=800.0 PL=0
MOVL C01578 V=800.0 PL=0
MOVL C01579 V=800.0 PL=0
MOVL C01580 V=800.0 PL=0
MOVL C01581 V=800.0 PL=0
MOVL C01582 V=800.0 PL=0
MOVL C01583 V=800.0 PL=0
MOVL C01584 V=800.0 PL=0
MOVL C01585 V=800.0 PL=0
MOVL C01586 V=800.0 PL=0
MOVL C01587 V=800.0 PL=0
MOVL C01588 V=800.0 PL=0
MOVL C01589 V=800.0 PL=0
MOVL C01590 V=800.0 PL=0
MOVL C01591 V=800.0 PL=0
MOVL C01592 V=800.0 PL=0
MOVL C01593 V=800.0 PL=0
MOVL C01594 V=800.0 PL=0
MOVL C01595 V=800.0 PL=0
MOVL C01596 V=800.0 PL=0
MOVL C01597 V=800.0 PL=0
MOVL C01598 V=800.0 PL=0
MOVL C01599 V=800.0 PL=0
MOVL C01600 V=800.0 PL=0
MOVL C01601 V=800.0 PL=0
MOVL C01602 V=800.0 PL=0
MOVL C01603 V=800.0 PL=0
MOVL C01604 V=800.0 PL=0
MOVL C01605 V=800.0 PL=0
MOVL C01606 V=800.0 PL=0
MOVL C01607 V=800.0 PL=0
MOVL C01608 V=800.0 PL=0
MOVL C01609 V=800.0 PL=0
MOVL C01610 V=800.0 PL=0
MOVL C01611 V=800.0 PL=0
MOVL C01612 V=800.0 PL=0
MOVL C01613 V=800.0 PL=0
MOVL C01614 V=800.0 PL=0
MOVL C01615 V=800.0 PL=0
MOVL C01616 V=800.0 PL=0
MOVL C01617 V=800.0 PL=0
MOVL C01618 V=800.0 PL=0
MOVL C01619 V=800.0 PL=0
MOVL C01620 V=800.0 PL=0
MOVL C01621 V=800.0 PL=0
MOVL C01622 V=800.0 PL=0
MOVL C01623 V=800.0 PL=0
MOVL C01624 V=800.0 PL=0
MOVL C01625 V=800.0 PL=0
MOVL C01626 V=800.0 PL=0
MOVL C01627 V=800.0 PL=0
MOVL C01628 V=800.0 PL=0
MOVL C01629 V=800.0 PL=0
MOVL C01630 V=800.0 PL=0
MOVL C01631 V=800.0 PL=0
MOVL C01632 V=800.0 PL=0
MOVL C01633 V=800.0 PL=0
MOVL C01634 V=800.0 PL=0
MOVL C01635 V=800.0 PL=0
MOVL C01636 V=800.0 PL=0
MOVL C01637 V=800.0 PL=0
MOVL C01638 V=800.0 PL=0
MOVL C01639 V=800.0 PL=0
MOVL C01640 V=800.0 PL=0
MOVL C01641 V=800.0 PL=0
MOVL C01642 V=800.0 PL=0
MOVL C01643 V=800.0 PL=0
MOVL C01644 V=800.0 PL=0
MOVL C01645 V=800.0 PL=0
MOVL C01646 V=800.0 PL=0
MOVL C01647 V=800.0 PL=0
MOVL C01648 V=800.0 PL=0
MOVL C01649 V=800.0 PL=0
MOVL C01650 V=800.0 PL=0
MOVL C01651 V=800.0 PL=0
MOVL C01652 V=800.0 PL=0
MOVL C01653 V=800.0 PL=0
MOVL C01654 V=800.0 PL=0
MOVL C01655 V=800.0 PL=0
MOVL C01656 V=800.0 PL=0
MOVL C01657 V=800.0 PL=0
MOVL C01658 V=800.0 PL=0
MOVL C01659 V=800.0 PL=0
MOVL C01660 V=800.0 PL=0
MOVL C01661 V=800.0 PL=0
MOVL C01662 V=800.0 PL=0
MOVL C01663 V=800.0 PL=0
MOVL C01664 V=800.0 PL=0
MOVL C01665 V=800.0 PL=0
MOVL C01666 V=800.0 PL=0
MOVL C01667 V=800.0 PL=0
MOVL C01668 V=800.0 PL=0
MOVL C01669 V=800.0 PL=0
MOVL C01670 V=800.0 PL=0
MOVL C01671 V=800.0 PL=0
MOVL C01672 V=800.0 PL=0
MOVL C01673 V=800.0 PL=0
MOVL C01674 V=800.0 PL=0
MOVL C01675 V=800.0 PL=0
MOVL C01676 V=800.0 PL=0
MOVL C01677 V=800.0 PL=0
MOVL C01678 V=800.0 PL=0
MOVL C01679 V=800.0 PL=0
MOVL C01680 V=800.0 PL=0
MOVL C01681 V=800.0 PL=0
MOVL C01682 V=800.0 PL=0
MOVL C01683 V=800.0 PL=0
MOVL C01684 V=800.0 PL=0
MOVL C01685 V=800.0 PL=0
MOVL C01686 V=800.0 PL=0
MOVL C01687 V=800.0 PL=0
MOVL C01688 V=800.0 PL=0
MOVL C01689 V=800.0 PL=0
MOVL C01690 V=800.0 PL=0
MOVL C01691 V=800.0 PL=0
MOVL C01692 V=800.0 PL=0
MOVL C01693 V=800.0 PL=0
MOVL C01694 V=800.0 PL=0
MOVL C01695 V=800.0 PL=0
MOVL C01696 V=800.0 PL=0
MOVL C01697 V=800.0 PL=0
MOVL C01698 V=800.0 PL=0
MOVL C01699 V=800.0 PL=0
MOVL C01700 V=800.0 PL=0
MOVL C01701 V=800.0 PL=0
MOVL C01702 V=800.0 PL=0
MOVL C01703 V=800.0 PL=0
MOVL C01704 V=800.0 PL=0
MOVL C01705 V=800.0 PL=0
MOVL C01706 V=800.0 PL=0
MOVL C01707 V=800.0 PL=0
MOVL C01708 V=800.0 PL=0
MOVL C01709 V=800.0 PL=0
MOVL C01710 V=800.0 PL=0
MOVL C01711 V=800.0 PL=0
MOVL C01712 V=800.0 PL=0
MOVL C01713 V=800.0 PL=0
MOVL C01714 V=800.0 PL=0
MOVL C01715 V=800.0 PL=0
MOVL C01716 V=800.0 PL=0
MOVL C01717 V=800.0 PL=0
MOVL C01718 V=800.0 PL=0
MOVL C01719 V=800.0 PL=0
MOVL C01720 V=800.0 PL=0
MOVL C01721 V=800.0 PL=0
MOVL C01722 V=800.0 PL=0
MOVL C01723 V=800.0 PL=0
MOVL C01724 V=800.0 PL=0
MOVL C01725 V=800.0 PL=0
MOVL C01726 V=800.0 PL=0
MOVL C01727 V=800.0 PL=0
MOVL C01728 V=800.0 PL=0
MOVL C01729 V=800.0 PL=0
MOVL C01730 V=800.0 PL=0
MOVL C01731 V=800.0 PL=0
MOVL C01732 V=800.0 PL=0
MOVL C01733 V=800.0 PL=0
MOVL C01734 V=800.0 PL=0
MOVL C01735 V=800.0 PL=0
MOVL C01736 V=800.0 PL=0
MOVL C01737 V=800.0 PL=0
MOVL C01738 V=800.0 PL=0
MOVL C01739 V=800.0 PL=0
MOVL C01740 V=800.0 PL=0
MOVL C01741 V=800.0 PL=0
MOVL C01742 V=800.0 PL=0
MOVL C01743 V=800.0 PL=0
MOVL C01744 V=800.0 PL=0
MOVL C01745 V=800.0 PL=0
MOVL C01746 V=800.0 PL=0
MOVL C01747 V=800.0 PL=0
MOVL C01748 V=800.0 PL=0
MOVL C01749 V=800.0 PL=0
MOVL C01750 V=800.0 PL=0
MOVL C01751 V=800.0 PL=0
MOVL C01752 V=800.0 PL=0
MOVL C01753 V=800.0 PL=0
MOVL C01754 V=800.0 PL=0
MOVL C01755 V=800.0 PL=0
MOVL C01756 V=800.0 PL=0
MOVL C01757 V=800.0 PL=0
MOVL C01758 V=800.0 PL=0
MOVL C01759 V=800.0 PL=0
MOVL C01760 V=800.0 PL=0
MOVL C01761 V=800.0 PL=0
MOVL C01762 V=800.0 PL=0
MOVL C01763 V=800.0 PL=0
MOVL C01764 V=800.0 PL=0
MOVL C01765 V=800.0 PL=0
MOVL C01766 V=800.0 PL=0
MOVL C01767 V=800.0 PL=0
MOVL C01768 V=800.0 PL=0
MOVL C01769 V=800.0 PL=0
MOVL C01770 V=800.0 PL=0
MOVL C01771 V=800.0 PL=0
MOVL C01772 V=800.0 PL=0
MOVL C01773 V=800.0 PL=0
MOVL C01774 V=800.0 PL=0
MOVL C01775 V=800.0 PL=0
MOVL C01776 V=800.0 PL=0
MOVL C01777 V=800.0 PL=0
MOVL C01778 V=800.0 PL=0
MOVL C01779 V=800.0 PL=0
MOVL C01780 V=800.0 PL=0
MOVL C01781 V=800.0 PL=0
MOVL C01782 V=800.0 PL=0
MOVL C01783 V=800.0 PL=0
MOVL C01784 V=800.0 PL=0
MOVL C01785 V=800.0 PL=0
MOVL C01786 V=800.0 PL=0
MOVL C01787 V=800.0 PL=0
MOVL C01788 V=800.0 PL=0
MOVL C01789 V=800.0 PL=0
MOVL C01790 V=800.0 PL=0
MOVL C01791 V=800.0 PL=0
MOVL C01792 V=800.0 PL=0
MOVL C01793 V=800.0 PL=0
MOVL C01794 V=800.0 PL=0
MOVL C01795 V=800.0 PL=0
MOVL C01796 V=800.0 PL=0
MOVL C01797 V=800.0 PL=0
MOVL C01798 V=800.0 PL=0
MOVL C01799 V=800.0 PL=0
MOVL C01800 V=800.0 PL=0
MOVL C01801 V=800.0 PL=0
MOVL C01802 V=800.0 PL=0
MOVL C01803 V=800.0 PL=0
MOVL C01804 V=800.0 PL=0
MOVL C01805 V=800.0 PL=0
MOVL C01806 V=800.0 PL=0
MOVL C01807 V=800.0 PL=0
MOVL C01808 V=800.0 PL=0
MOVL C01809 V=800.0 PL=0
MOVL C01810 V=800.0 PL=0
MOVL C01811 V=800.0 PL=0
MOVL C01812 V=800.0 PL=0
MOVL C01813 V=800.0 PL=0
MOVL C01814 V=800.0 PL=0
MOVL C01815 V=800.0 PL=0
MOVL C01816 V=800.0 PL=0
MOVL C01817 V=800.0 PL=0
MOVL C01818 V=800.0 PL=0
MOVL C01819 V=800.0 PL=0
MOVL C01820 V=800.0 PL=0
MOVL C01821 V=800.0 PL=0
MOVL C01822 V=800.0 PL=0
MOVL C01823 V=800.0 PL=0
MOVL C01824 V=800.0 PL=0
MOVL C01825 V=800.0 PL=0
MOVL C01826 V=800.0 PL=0
MOVL C01827 V=800.0 PL=0
MOVL C01828 V=800.0 PL=0
MOVL C01829 V=800.0 PL=0
MOVL C01830 V=800.0 PL=0
MOVL C01831 V=800.0 PL=0
MOVL C01832 V=800.0 PL=0
MOVL C01833 V=800.0 PL=0
MOVL C01834 V=800.0 PL=0
MOVL C01835 V=800.0 PL=0
MOVL C01836 V=800.0 PL=0
MOVL C01837 V=800.0 PL=0
MOVL C01838 V=800.0 PL=0
MOVL C01839 V=800.0 PL=0
MOVL C01840 V=800.0 PL=0
MOVL C01841 V=800.0 PL=0
MOVL C01842 V=800.0 PL=0
MOVL C01843 V=800.0 PL=0
MOVL C01844 V=800.0 PL=0
MOVL C01845 V=800.0 PL=0
MOVL C01846 V=800.0 PL=0
MOVL C01847 V=800.0 PL=0
MOVL C01848 V=800.0 PL=0
MOVL C01849 V=800.0 PL=0
MOVL C01850 V=800.0 PL=0
MOVL C01851 V=800.0 PL=0
MOVL C01852 V=800.0 PL=0
MOVL C01853 V=800.0 PL=0
MOVL C01854 V=800.0 PL=0
MOVL C01855 V=800.0 PL=0
MOVL C01856 V=800.0 PL=0
MOVL C01857 V=800.0 PL=0
MOVL C01858 V=800.0 PL=0
MOVL C01859 V=800.0 PL=0
MOVL C01860 V=800.0 PL=0
MOVL C01861 V=800.0 PL=0
MOVL C01862 V=800.0 PL=0
MOVL C01863 V=800.0 PL=0
MOVL C01864 V=800.0 PL=0
MOVL C01865 V=800.0 PL=0
MOVL C01866 V=800.0 PL=0
MOVL C01867 V=800.0 PL=0
MOVL C01868 V=800.0 PL=0
MOVL C01869 V=800.0 PL=0
MOVL C01870 V=800.0 PL=0
MOVL C01871 V=800.0 PL=0
MOVL C01872 V=800.0 PL=0
MOVL C01873 V=800.0 PL=0
MOVL C01874 V=800.0 PL=0
MOVL C01875 V=800.0 PL=0
MOVL C01876 V=800.0 PL=0
MOVL C01877 V=800.0 PL=0
MOVL C01878 V=800.0 PL=0
MOVL C01879 V=800.0 PL=0
MOVL C01880 V=800.0 PL=0
MOVL C01881 V=800.0 PL=0
MOVL C01882 V=800.0 PL=0
MOVL C01883 V=800.0 PL=0
MOVL C01884 V=800.0 PL=0
MOVL C01885 V=800.0 PL=0
MOVL C01886 V=800.0 PL=0
MOVL C01887 V=800.0 PL=0
MOVL C01888 V=800.0 PL=0
MOVL C01889 V=800.0 PL=0
MOVL C01890 V=800.0 PL=0
MOVL C01891 V=800.0 PL=0
MOVL C01892 V=800.0 PL=0
MOVL C01893 V=800.0 PL=0
MOVL C01894 V=800.0 PL=0
MOVL C01895 V=800.0 PL=0
MOVL C01896 V=800.0 PL=0
MOVL C01897 V=800.0 PL=0
MOVL C01898 V=800.0 PL=0
MOVL C01899 V=800.0 PL=0
MOVL C01900 V=800.0 PL=0
MOVL C01901 V=800.0 PL=0
MOVL C01902 V=800.0 PL=0
MOVL C01903 V=800.0 PL=0
MOVL C01904 V=800.0 PL=0
MOVL C01905 V=800.0 PL=0
MOVL C01906 V=800.0 PL=0
MOVL C01907 V=800.0 PL=0
MOVL C01908 V=800.0 PL=0
MOVL C01909 V=800.0 PL=0
MOVL C01910 V=800.0 PL=0
MOVL C01911 V=800.0 PL=0
MOVL C01912 V=800.0 PL=0
MOVL C01913 V=800.0 PL=0
MOVL C01914 V=800.0 PL=0
MOVL C01915 V=800.0 PL=0
MOVL C01916 V=800.0 PL=0
MOVL C01917 V=800.0 PL=0
MOVL C01918 V=800.0 PL=0
MOVL C01919 V=800.0 PL=0
MOVL C01920 V=800.0 PL=0
MOVL C01921 V=800.0 PL=0
MOVL C01922 V=800.0 PL=0
MOVL C01923 V=800.0 PL=0
MOVL C01924 V=800.0 PL=0
MOVL C01925 V=800.0 PL=0
MOVL C01926 V=800.0 PL=0
MOVL C01927 V=800.0 PL=0
MOVL C01928 V=800.0 PL=0
MOVL C01929 V=800.0 PL=0
MOVL C01930 V=800.0 PL=0
MOVL C01931 V=800.0 PL=0
MOVL C01932 V=800.0 PL=0
MOVL C01933 V=800.0 PL=0
MOVL C01934 V=800.0 PL=0
MOVL C01935 V=800.0 PL=0
MOVL C01936 V=800.0 PL=0
MOVL C01937 V=800.0 PL=0
MOVL C01938 V=800.0 PL=0
MOVL C01939 V=800.0 PL=0
MOVL C01940 V=800.0 PL=0
MOVL C01941 V=800.0 PL=0
MOVL C01942 V=800.0 PL=0
MOVL C01943 V=800.0 PL=0
MOVL C01944 V=800.0 PL=0
MOVL C01945 V=800.0 PL=0
MOVL C01946 V=800.0 PL=0
MOVL C01947 V=800.0 PL=0
MOVL C01948 V=800.0 PL=0
MOVL C01949 V=800.0 PL=0
MOVL C01950 V=800.0 PL=0
MOVL C01951 V=800.0 PL=0
MOVL C01952 V=800.0 PL=0
MOVL C01953 V=800.0 PL=0
MOVL C01954 V=800.0 PL=0
MOVL C01955 V=800.0 PL=0
MOVL C01956 V=800.0 PL=0
MOVL C01957 V=800.0 PL=0
MOVL C01958 V=800.0 PL=0
MOVL C01959 V=800.0 PL=0
MOVL C01960 V=800.0 PL=0
MOVL C01961 V=800.0 PL=0
MOVL C01962 V=800.0 PL=0
MOVL C01963 V=800.0 PL=0
MOVL C01964 V=800.0 PL=0
MOVL C01965 V=800.0 PL=0
MOVL C01966 V=800.0 PL=0
MOVL C01967 V=800.0 PL=0
MOVL C01968 V=800.0 PL=0
MOVL C01969 V=800.0 PL=0
MOVL C01970 V=800.0 PL=0
MOVL C01971 V=800.0 PL=0
MOVL C01972 V=800.0 PL=0
MOVL C01973 V=800.0 PL=0
MOVL C01974 V=800.0 PL=0
MOVL C01975 V=800.0 PL=0
MOVL C01976 V=800.0 PL=0
MOVL C01977 V=800.0 PL=0
MOVL C01978 V=800.0 PL=0
MOVL C01979 V=800.0 PL=0
MOVL C01980 V=800.0 PL=0
MOVL C01981 V=800.0 PL=0
MOVL C01982 V=800.0 PL=0
MOVL C01983 V=800.0 PL=0
MOVL C01984 V=800.0 PL=0
MOVL C01985 V=800.0 PL=0
MOVL C01986 V=800.0 PL=0
MOVL C01987 V=800.0 PL=0
MOVL C01988 V=800.0 PL=0
MOVL C01989 V=800.0 PL=0
MOVL C01990 V=800.0 PL=0
MOVL C01991 V=800.0 PL=0
MOVL C01992 V=800.0 PL=0
MOVL C01993 V=800.0 PL=0
MOVL C01994 V=800.0 PL=0
MOVL C01995 V=800.0 PL=0
MOVL C01996 V=800.0 PL=0
MOVL C01997 V=800.0 PL=0
MOVL C01998 V=800.0 PL=0
MOVL C01999 V=800.0 PL=0
MOVL C02000 V=800.0 PL=0
MOVL C02001 V=800.0 PL=0
MOVL C02002 V=800.0 PL=0
MOVL C02003 V=800.0 PL=0
MOVL C02004 V=800.0 PL=0
MOVL C02005 V=800.0 PL=0
MOVL C02006 V=800.0 PL=0
MOVL C02007 V=800.0 PL=0
MOVL C02008 V=800.0 PL=0
MOVL C02009 V=800.0 PL=0
MOVL C02010 V=800.0 PL=0
MOVL C02011 V=800.0 PL=0
MOVL C02012 V=800.0 PL=0
MOVL C02013 V=800.0 PL=0
MOVL C02014 V=800.0 PL=0
MOVL C02015 V=800.0 PL=0
MOVL C02016 V=800.0 PL=0
MOVL C02017 V=800.0 PL=0
MOVL C02018 V=800.0 PL=0
MOVL C02019 V=800.0 PL=0
MOVL C02020 V=800.0 PL=0
MOVL C02021 V=800.0 PL=0
MOVL C02022 V=800.0 PL=0
MOVL C02023 V=800.0 PL=0
MOVL C02024 V=800.0 PL=0
MOVL C02025 V=800.0 PL=0
MOVL C02026 V=800.0 PL=0
MOVL C02027 V=800.0 PL=0
MOVL C02028 V=800.0 PL=0
MOVL C02029 V=800.0 PL=0
MOVL C02030 V=800.0 PL=0
MOVL C02031 V=800.0 PL=0
MOVL C02032 V=800.0 PL=0
MOVL C02033 V=800.0 PL=0
MOVL C02034 V=800.0 PL=0
MOVL C02035 V=800.0 PL=0
MOVL C02036 V=800.0 PL=0
MOVL C02037 V=800.0 PL=0
MOVL C02038 V=800.0 PL=0
MOVL C02039 V=800.0 PL=0
MOVL C02040 V=800.0 PL=0
MOVL C02041 V=800.0 PL=0
MOVL C02042 V=800.0 PL=0
MOVL C02043 V=800.0 PL=0
MOVL C02044 V=800.0 PL=0
MOVL C02045 V=800.0 PL=0
MOVL C02046 V=800.0 PL=0
MOVL C02047 V=800.0 PL=0
MOVL C02048 V=800.0 PL=0
MOVL C02049 V=800.0 PL=0
MOVL C02050 V=800.0 PL=0
MOVL C02051 V=800.0 PL=0
MOVL C02052 V=800.0 PL=0
MOVL C02053 V=800.0 PL=0
MOVL C02054 V=800.0 PL=0
MOVL C02055 V=800.0 PL=0
MOVL C02056 V=800.0 PL=0
MOVL C02057 V=800.0 PL=0
MOVL C02058 V=800.0 PL=0
MOVL C02059 V=800.0 PL=0
MOVL C02060 V=800.0 PL=0
MOVL C02061 V=800.0 PL=0
MOVL C02062 V=800.0 PL=0
MOVL C02063 V=800.0 PL=0
MOVL C02064 V=800.0 PL=0
MOVL C02065 V=800.0 PL=0
MOVL C02066 V=800.0 PL=0
MOVL C02067 V=800.0 PL=0
MOVL C02068 V=800.0 PL=0
MOVL C02069 V=800.0 PL=0
MOVL C02070 V=800.0 PL=0
MOVL C02071 V=800.0 PL=0
MOVL C02072 V=800.0 PL=0
MOVL C02073 V=800.0 PL=0
MOVL C02074 V=800.0 PL=0
MOVL C02075 V=800.0 PL=0
MOVL C02076 V=800.0 PL=0
MOVL C02077 V=800.0 PL=0
MOVL C02078 V=800.0 PL=0
MOVL C02079 V=800.0 PL=0
MOVL C02080 V=800.0 PL=0
MOVL C02081 V=800.0 PL=0
MOVL C02082 V=800.0 PL=0
MOVL C02083 V=800.0 PL=0
MOVL C02084 V=800.0 PL=0
MOVL C02085 V=800.0 PL=0
MOVL C02086 V=800.0 PL=0
MOVL C02087 V=800.0 PL=0
MOVL C02088 V=800.0 PL=0
MOVL C02089 V=800.0 PL=0
MOVL C02090 V=800.0 PL=0
MOVL C02091 V=800.0 PL=0
MOVL C02092 V=800.0 PL=0
MOVL C02093 V=800.0 PL=0
MOVL C02094 V=800.0 PL=0
MOVL C02095 V=800.0 PL=0
MOVL C02096 V=800.0 PL=0
MOVL C02097 V=800.0 PL=0
MOVL C02098 V=800.0 PL=0
MOVL C02099 V=800.0 PL=0
MOVL C02100 V=800.0 PL=0
MOVL C02101 V=800.0 PL=0
MOVL C02102 V=800.0 PL=0
MOVL C02103 V=800.0 PL=0
MOVL C02104 V=800.0 PL=0
MOVL C02105 V=800.0 PL=0
MOVL C02106 V=800.0 PL=0
MOVL C02107 V=800.0 PL=0
MOVL C02108 V=800.0 PL=0
MOVL C02109 V=800.0 PL=0
MOVL C02110 V=800.0 PL=0
MOVL C02111 V=800.0 PL=0
MOVL C02112 V=800.0 PL=0
MOVL C02113 V=800.0 PL=0
MOVL C02114 V=800.0 PL=0
MOVL C02115 V=800.0 PL=0
MOVL C02116 V=800.0 PL=0
MOVL C02117 V=800.0 PL=0
MOVL C02118 V=800.0 PL=0
MOVL C02119 V=800.0 PL=0
MOVL C02120 V=800.0 PL=0
MOVL C02121 V=800.0 PL=0
MOVL C02122 V=800.0 PL=0
MOVL C02123 V=800.0 PL=0
MOVL C02124 V=800.0 PL=0
MOVL C02125 V=800.0 PL=0
MOVL C02126 V=800.0 PL=0
MOVL C02127 V=800.0 PL=0
MOVL C02128 V=800.0 PL=0
MOVL C02129 V=800.0 PL=0
MOVL C02130 V=800.0 PL=0
MOVL C02131 V=800.0 PL=0
MOVL C02132 V=800.0 PL=0
MOVL C02133 V=800.0 PL=0
MOVL C02134 V=800.0 PL=0
MOVL C02135 V=800.0 PL=0
MOVL C02136 V=800.0 PL=0
MOVL C02137 V=800.0 PL=0
MOVL C02138 V=800.0 PL=0
MOVL C02139 V=800.0 PL=0
MOVL C02140 V=800.0 PL=0
MOVL C02141 V=800.0 PL=0
MOVL C02142 V=800.0 PL=0
MOVL C02143 V=800.0 PL=0
MOVL C02144 V=800.0 PL=0
MOVL C02145 V=800.0 PL=0
MOVL C02146 V=800.0 PL=0
MOVL C02147 V=800.0 PL=0
MOVL C02148 V=800.0 PL=0
MOVL C02149 V=800.0 PL=0
